(* IEC 61131-3 sources: ics-sorter-range/, 2 files *)

(* ---- Sorter.st ---- *)
(* Three-lane matrix sorter with nine trailer doors.
   Generated by gen_sorter.py. Do not hand edit; regenerate instead. *)

TYPE
  BELT_T : ARRAY[0..19] OF INT;
END_TYPE

PROGRAM sorter
VAR
  sorter_run    AT %QX110.0    : BOOL;   (* operator master run *)
  auto_mode     AT %QX110.1    : BOOL;   (* auto routing enabled *)
  lane1_run     AT %QX110.2    : BOOL;   (* induct 1 running *)
  lane2_run     AT %QX110.3    : BOOL;   (* induct 2 running *)
  lane3_run     AT %QX110.4    : BOOL;   (* induct 3 running *)
  ob1_run       AT %QX110.5    : BOOL;   (* outbound 1 running *)
  ob2_run       AT %QX110.6    : BOOL;   (* outbound 2 running *)
  ob3_run       AT %QX110.7    : BOOL;   (* outbound 3 running *)
  l1_div1       AT %QX111.0    : BOOL;   (* lane 1 divert to outbound 1 *)
  l1_div2       AT %QX111.1    : BOOL;   (* lane 1 divert to outbound 2 *)
  l1_div3       AT %QX111.2    : BOOL;   (* lane 1 divert to outbound 3 *)
  l2_div1       AT %QX111.3    : BOOL;   (* lane 2 divert to outbound 1 *)
  l2_div2       AT %QX111.4    : BOOL;   (* lane 2 divert to outbound 2 *)
  l2_div3       AT %QX111.5    : BOOL;   (* lane 2 divert to outbound 3 *)
  l3_div1       AT %QX111.6    : BOOL;   (* lane 3 divert to outbound 1 *)
  l3_div2       AT %QX111.7    : BOOL;   (* lane 3 divert to outbound 2 *)
  l3_div3       AT %QX112.0    : BOOL;   (* lane 3 divert to outbound 3 *)
  b1_door1      AT %QX112.1    : BOOL;   (* outbound 1 divert to door 1 *)
  b1_door2      AT %QX112.2    : BOOL;   (* outbound 1 divert to door 2 *)
  b1_door3      AT %QX112.3    : BOOL;   (* outbound 1 divert to door 3 *)
  b2_door1      AT %QX112.4    : BOOL;   (* outbound 2 divert to door 1 *)
  b2_door2      AT %QX112.5    : BOOL;   (* outbound 2 divert to door 2 *)
  b2_door3      AT %QX112.6    : BOOL;   (* outbound 2 divert to door 3 *)
  b3_door1      AT %QX112.7    : BOOL;   (* outbound 3 divert to door 1 *)
  b3_door2      AT %QX113.0    : BOOL;   (* outbound 3 divert to door 2 *)
  b3_door3      AT %QX113.1    : BOOL;   (* outbound 3 divert to door 3 *)
  jam_alarm     AT %QX113.2    : BOOL;   (* induct belt backing up at the tail *)
  coll_alarm    AT %QX113.3    : BOOL;   (* merge collision on an outbound belt *)
  noread_alarm  AT %QX113.4    : BOOL;   (* tunnel no-read *)
  nohome_alarm  AT %QX113.5    : BOOL;   (* package reached end of an outbound belt *)
  reset_cmd     AT %QX113.6    : BOOL;   (* re-run the init block, clearing all process state *)
  fault_reset   AT %QX113.7    : BOOL;   (* hold the drive fault-reset bit for several scans *)
  scanner_fault_ack AT %QX114.0 : BOOL; (* operator acknowledges scanner fault *)
  scanner_retry AT %QX114.1 : BOOL;     (* operator retries after acknowledgement *)
  xle_mode AT %QX114.2 : BOOL;           (* lane 1 external sort decisions *)
  xle_multi AT %QX114.3 : BOOL;          (* bounded two-package external mode *)
  plant_mode AT %QX114.6 : BOOL;          (* lane 1 position comes from drives plant *)
  photoeye_mode AT %QX114.7 : BOOL;       (* opt-in stateful field inputs; legacy events remain *)
  accumulation_mode AT %QX115.0 : BOOL;   (* opt-in finite plant zones; coil 920 *)

  speed_sp_1    AT %QW200      : INT;    (* induct 1 speed setpoint, rpm *)
  speed_sp_2    AT %QW201      : INT;    (* induct 2 speed setpoint, rpm *)
  speed_sp_3    AT %QW202      : INT;    (* induct 3 speed setpoint, rpm *)
  ob_speed_1    AT %QW203      : INT;    (* outbound 1 speed setpoint, rpm *)
  ob_speed_2    AT %QW204      : INT;    (* outbound 2 speed setpoint, rpm *)
  ob_speed_3    AT %QW205      : INT;    (* outbound 3 speed setpoint, rpm *)
  min_gap_sp    AT %QW206      : INT;    (* minimum induct gap, cells *)
  rate_sp_1     AT %QW207      : INT;    (* induct 1 interval, scans per package *)
  rate_sp_2     AT %QW208      : INT;    (* induct 2 interval, scans per package *)
  rate_sp_3     AT %QW209      : INT;    (* induct 3 interval, scans per package *)
  noread_sp     AT %QW210      : INT;    (* tunnel no-read rate, per mille *)
  scan_code_1   AT %QW211      : INT;    (* last barcode read by tunnel 1 *)
  scan_code_2   AT %QW212      : INT;    (* last barcode read by tunnel 2 *)
  scan_code_3   AT %QW213      : INT;    (* last barcode read by tunnel 3 *)
  noread_ct     AT %QW214      : INT;    (* cumulative tunnel no-reads *)
  coll_ct       AT %QW215      : INT;    (* cumulative merge collisions *)
  jam_ct        AT %QW216      : INT;    (* cumulative induct belt jams *)
  missort_ct    AT %QW217      : INT;    (* cumulative confirmed missorts at door scan *)
  recirc_ct     AT %QW218      : INT;    (* packages undiverted off an induct belt *)
  nohome_ct     AT %QW219      : INT;    (* packages undiverted off an outbound belt *)
  inducted_ct   AT %QW220      : INT;    (* cumulative packages inducted *)
  serial_next   AT %QW221      : INT;    (* next package serial number *)
  tr11_ct       AT %QW222      : INT;    (* packages loaded to trailer 1-1 *)
  tr12_ct       AT %QW223      : INT;    (* packages loaded to trailer 1-2 *)
  tr13_ct       AT %QW224      : INT;    (* packages loaded to trailer 1-3 *)
  tr21_ct       AT %QW225      : INT;    (* packages loaded to trailer 2-1 *)
  tr22_ct       AT %QW226      : INT;    (* packages loaded to trailer 2-2 *)
  tr23_ct       AT %QW227      : INT;    (* packages loaded to trailer 2-3 *)
  tr31_ct       AT %QW228      : INT;    (* packages loaded to trailer 3-1 *)
  tr32_ct       AT %QW229      : INT;    (* packages loaded to trailer 3-2 *)
  tr33_ct       AT %QW230      : INT;    (* packages loaded to trailer 3-3 *)
  tr11_bad      AT %QW231      : INT;    (* wrong-destination loads at trailer 1-1 *)
  tr12_bad      AT %QW232      : INT;    (* wrong-destination loads at trailer 1-2 *)
  tr13_bad      AT %QW233      : INT;    (* wrong-destination loads at trailer 1-3 *)
  tr21_bad      AT %QW234      : INT;    (* wrong-destination loads at trailer 2-1 *)
  tr22_bad      AT %QW235      : INT;    (* wrong-destination loads at trailer 2-2 *)
  tr23_bad      AT %QW236      : INT;    (* wrong-destination loads at trailer 2-3 *)
  tr31_bad      AT %QW237      : INT;    (* wrong-destination loads at trailer 3-1 *)
  tr32_bad      AT %QW238      : INT;    (* wrong-destination loads at trailer 3-2 *)
  tr33_bad      AT %QW239      : INT;    (* wrong-destination loads at trailer 3-3 *)
  div_act_1     AT %QW240      : INT;    (* outbound 1 induct-divert actuations *)
  div_act_2     AT %QW241      : INT;    (* outbound 2 induct-divert actuations *)
  div_act_3     AT %QW242      : INT;    (* outbound 3 induct-divert actuations *)
  scan_ct       AT %QW243      : INT;    (* PLC scans since init, logical clock *)
  shift_ct_1    AT %QW244      : INT;    (* induct 1 belt shifts since init *)
  shift_ct_2    AT %QW245      : INT;    (* induct 2 belt shifts since init *)
  shift_ct_3    AT %QW246      : INT;    (* induct 3 belt shifts since init *)
  master_seed   AT %QW247      : INT;    (* PRNG root, 1..999, 0 means use default *)
  run_id        AT %QW248      : INT;    (* scenario run identifier, echoed into telemetry *)
  prog_hash     AT %QW249      : INT;    (* identity of the generated program, set at init *)
  multiple_ct   AT %QW250      : INT;    (* tunnel reported more than one barcode *)
  oversize_ct   AT %QW251      : INT;    (* package exceeded the tunnel size limit *)
  duplicate_ct  AT %QW252      : INT;    (* tunnel returned a barcode already seen *)
  invalid_ct    AT %QW253      : INT;    (* tunnel decoded something that is not a label *)
  scan_late_ct  AT %QW254      : INT;    (* package left the tunnel before its result arrived *)
  scanner_state AT %QW255 : INT;        (* 0 ready, 1 prepare, 2 reset, 3 fault, 4 acknowledged *)
  scanner_fault_mask AT %QW256 : INT;   (* bits 0,1,2 identify missing tunnel ACKs *)
  scanner_ack_mask AT %QW257 : INT;     (* bits 0,1,2 for current phase ACKs *)
  scanner_wait AT %QW258 : INT;         (* elapsed PLC scans in current phase *)
  xle_cmd_id AT %QW500 : INT;            (* XLe writes 500..503 *)
  xle_cmd_bc AT %QW501 : INT;
  xle_cmd_dest AT %QW502 : INT;
  xle_cmd_nonce AT %QW503 : INT;
  xle_ack_id AT %QW504 : INT;            (* PLC writes 504..509 *)
  xle_state AT %QW505 : INT;             (* 0 idle, 1 accepted, 2 diverted, 3 loaded, 4 failed, 5 recirc *)
  xle_reason AT %QW506 : INT;            (* 1 no decision, 2 invalid/late, 3 collision, 4 no home, 5 wrong door *)
  xle_actual AT %QW507 : INT;            (* physical trailer, 1..9 *)
  xle_package AT %QW508 : INT;           (* scanner barcode identity *)
  xle_run_nonce AT %QW509 : INT;
  xle_scan_tick AT %QW510 : INT;          (* PLC scan accepting tunnel 1 result *)
  xle_accept_tick AT %QW511 : INT;        (* PLC scan accepting XLe command *)
  xle_divert_tick AT %QW512 : INT;        (* first arrival at lane 1 cell 14 *)
  multi_op AT %QW520 : INT;              (* 1 route, 2 release terminal slot *)
  multi_slot AT %QW521 : INT;            (* slot index 0..2 *)
  multi_token AT %QW522 : INT;
  multi_serial AT %QW523 : INT;
  multi_seq AT %QW524 : INT;
  multi_bc AT %QW525 : INT;
  multi_dest AT %QW526 : INT;
  multi_nonce AT %QW527 : INT;
  multi_cmd_id AT %QW528 : INT;          (* write last; changed ID commits payload *)
  multi_ack AT %QW529 : INT;             (* 1 accepted, 2 rejected, 3 released *)
  slot0_token AT %QW530 : INT;
  slot0_serial AT %QW531 : INT;
  slot0_seq AT %QW532 : INT;
  slot0_bc AT %QW533 : INT;
  slot0_state AT %QW534 : INT;
  slot0_dest AT %QW535 : INT;
  slot0_actual AT %QW536 : INT;
  slot0_reason AT %QW537 : INT;
  slot0_scan AT %QW538 : INT;
  slot0_accept AT %QW539 : INT;
  slot0_divert AT %QW540 : INT;
  slot0_command AT %QW541 : INT;
  slot1_token AT %QW542 : INT;
  slot1_serial AT %QW543 : INT;
  slot1_seq AT %QW544 : INT;
  slot1_bc AT %QW545 : INT;
  slot1_state AT %QW546 : INT;
  slot1_dest AT %QW547 : INT;
  slot1_actual AT %QW548 : INT;
  slot1_reason AT %QW549 : INT;
  slot1_scan AT %QW550 : INT;
  slot1_accept AT %QW551 : INT;
  slot1_divert AT %QW552 : INT;
  slot1_command AT %QW553 : INT;
  multi_ack_id AT %QW554 : INT;         (* PLC echoes processed command ID *)
  epoch_offer_lo AT %QW555 : INT;       (* XLe durable run ID, base 30000 *)
  epoch_offer_hi AT %QW556 : INT;
  epoch_offer_id AT %QW557 : INT;       (* write last to commit offer *)
  epoch_active_lo AT %QW558 : INT;      (* PLC accepted run ID *)
  epoch_active_hi AT %QW559 : INT;
  epoch_ack_id AT %QW560 : INT;
  epoch_fault AT %QW561 : INT;          (* 0 ready, 1 no identity, 2 XLe fault *)
  cmd_epoch_lo AT %QW562 : INT;
  cmd_epoch_hi AT %QW563 : INT;
  epoch_fault_request AT %QW564 : INT;  (* XLe 2 = fail closed *)
  hb_epoch_lo AT %QW565 : INT;          (* heartbeat payload before sequence *)
  hb_epoch_hi AT %QW566 : INT;
  hb_sequence AT %QW567 : INT;          (* XLe changes at least every 5 s *)
  hb_age AT %QW568 : INT;               (* PLC scans since valid heartbeat *)
  xle_liveness AT %QW569 : INT;         (* 0 healthy, 1 lost, 2 seen, 3 retry *)
  recovery_epoch_lo AT %QW570 : INT;
  recovery_epoch_hi AT %QW571 : INT;
  recovery_sequence AT %QW572 : INT;   (* XLe writes after journal verification *)
  hb_ack_sequence AT %QW573 : INT;
  plant_request AT %QW574 : INT;         (* PLC commits induction request last *)
  plant_request_token AT %QW575 : INT;
  plant_request_serial AT %QW576 : INT;
  plant_request_lane AT %QW577 : INT;   (* 1..3; written before request commit *)
  plant_event_lane AT %QW578 : INT;     (* plant payload, written before event commit *)
  plant_event_type AT %QW580 : INT;      (* 1 induct, 2 tunnel, 3 divert, 4 trailer, 5 recirc, 6 failed confirmation *)
  plant_event_token AT %QW581 : INT;
  plant_event_serial AT %QW582 : INT;
  plant_event_actual AT %QW583 : INT;    (* outbound 1..3 or trailer 1..9 *)
  plant_event_position AT %QW584 : INT;  (* tenths of a cell, telemetry *)
  plant_event_seq AT %QW585 : INT;       (* plant commits event last *)
  plant_event_ack AT %QW586 : INT;       (* PLC acknowledges even rejected events *)
  plant_epoch_lo AT %QW587 : INT;
  plant_epoch_hi AT %QW588 : INT;
  plant_nonce AT %QW589 : INT;
  plant_heartbeat AT %QW590 : INT;
  plant_fault AT %QW591 : INT;          (* 0 ready, 1 unavailable, 2 identity mismatch, 3 bad event *)
  plant_failed_count AT %QW592 : INT;   (* latched failed physical confirmations, cleared by reset *)
  plant_heartbeat_age AT %QW593 : INT;  (* PLC scans since the last plant heartbeat *)
  p0_raw_epoch_lo AT %QW600 : INT;
  p0_raw_epoch_hi AT %QW601 : INT;
  p0_raw_nonce AT %QW602 : INT;
  p0_raw_token AT %QW603 : INT;
  p0_raw_serial AT %QW604 : INT;
  p0_raw_belt AT %QW605 : INT;
  p0_raw_pos AT %QW606 : INT;
  p0_raw_event AT %QW607 : INT;
  p0_raw_actual AT %QW608 : INT;
  p0_raw_seq AT %QW609 : INT;
  p1_raw_epoch_lo AT %QW610 : INT;
  p1_raw_epoch_hi AT %QW611 : INT;
  p1_raw_nonce AT %QW612 : INT;
  p1_raw_token AT %QW613 : INT;
  p1_raw_serial AT %QW614 : INT;
  p1_raw_belt AT %QW615 : INT;
  p1_raw_pos AT %QW616 : INT;
  p1_raw_event AT %QW617 : INT;
  p1_raw_actual AT %QW618 : INT;
  p1_raw_seq AT %QW619 : INT;
  p0_view_epoch_lo AT %QW620 : INT;
  p0_view_epoch_hi AT %QW621 : INT;
  p0_view_nonce AT %QW622 : INT;
  p0_view_token AT %QW623 : INT;
  p0_view_serial AT %QW624 : INT;
  p0_view_belt AT %QW625 : INT;
  p0_view_pos AT %QW626 : INT;
  p0_view_event AT %QW627 : INT;
  p0_view_actual AT %QW628 : INT;
  p0_view_seq AT %QW629 : INT;
  p1_view_epoch_lo AT %QW630 : INT;
  p1_view_epoch_hi AT %QW631 : INT;
  p1_view_nonce AT %QW632 : INT;
  p1_view_token AT %QW633 : INT;
  p1_view_serial AT %QW634 : INT;
  p1_view_belt AT %QW635 : INT;
  p1_view_pos AT %QW636 : INT;
  p1_view_event AT %QW637 : INT;
  p1_view_actual AT %QW638 : INT;
  p1_view_seq AT %QW639 : INT;
  p0_view_status AT %QW640 : INT;       (* 0 empty, 1 live, 2 stale, 3 identity mismatch *)
  p1_view_status AT %QW641 : INT;
  p0_view_age AT %QW642 : INT;
  p1_view_age AT %QW643 : INT;
  slot0_lane AT %QW644 : INT;           (* stable lane identity beside slot row *)
  slot1_lane AT %QW645 : INT;
  plant_failed_lane AT %QW646 : INT;    (* lane of latest failed confirmation *)
  slot2_token AT %QW647 : INT;
  slot2_serial AT %QW648 : INT;
  slot2_seq AT %QW649 : INT;
  slot2_bc AT %QW650 : INT;
  slot2_state AT %QW651 : INT;
  slot2_dest AT %QW652 : INT;
  slot2_actual AT %QW653 : INT;
  slot2_reason AT %QW654 : INT;
  slot2_scan AT %QW655 : INT;
  slot2_accept AT %QW656 : INT;
  slot2_divert AT %QW657 : INT;
  slot2_command AT %QW658 : INT;
  slot2_lane AT %QW659 : INT;
  p2_raw_epoch_lo AT %QW660 : INT;
  p2_raw_epoch_hi AT %QW661 : INT;
  p2_raw_nonce AT %QW662 : INT;
  p2_raw_token AT %QW663 : INT;
  p2_raw_serial AT %QW664 : INT;
  p2_raw_belt AT %QW665 : INT;
  p2_raw_pos AT %QW666 : INT;
  p2_raw_event AT %QW667 : INT;
  p2_raw_actual AT %QW668 : INT;
  p2_raw_seq AT %QW669 : INT;
  p2_view_epoch_lo AT %QW670 : INT;
  p2_view_epoch_hi AT %QW671 : INT;
  p2_view_nonce AT %QW672 : INT;
  p2_view_token AT %QW673 : INT;
  p2_view_serial AT %QW674 : INT;
  p2_view_belt AT %QW675 : INT;
  p2_view_pos AT %QW676 : INT;
  p2_view_event AT %QW677 : INT;
  p2_view_actual AT %QW678 : INT;
  p2_view_seq AT %QW679 : INT;
  p2_view_status AT %QW680 : INT;
  p2_view_age AT %QW681 : INT;
  pe0_raw_epoch_lo AT %QW690 : INT;
  pe0_raw_epoch_hi AT %QW691 : INT;
  pe0_raw_nonce AT %QW692 : INT;
  pe0_raw_token AT %QW693 : INT;
  pe0_raw_serial AT %QW694 : INT;
  pe0_raw_lane AT %QW695 : INT;
  pe0_raw_mask AT %QW696 : INT;          (* bits 0..4: induct,tunnel,divert,outbound,trailer *)
  pe0_raw_seq AT %QW697 : INT;           (* plant commits the complete row last *)
  pe1_raw_epoch_lo AT %QW698 : INT;
  pe1_raw_epoch_hi AT %QW699 : INT;
  pe1_raw_nonce AT %QW700 : INT;
  pe1_raw_token AT %QW701 : INT;
  pe1_raw_serial AT %QW702 : INT;
  pe1_raw_lane AT %QW703 : INT;
  pe1_raw_mask AT %QW704 : INT;
  pe1_raw_seq AT %QW705 : INT;
  pe2_raw_epoch_lo AT %QW706 : INT;
  pe2_raw_epoch_hi AT %QW707 : INT;
  pe2_raw_nonce AT %QW708 : INT;
  pe2_raw_token AT %QW709 : INT;
  pe2_raw_serial AT %QW710 : INT;
  pe2_raw_lane AT %QW711 : INT;
  pe2_raw_mask AT %QW712 : INT;
  pe2_raw_seq AT %QW713 : INT;
  pe0_view_epoch_lo AT %QW720 : INT;
  pe0_view_epoch_hi AT %QW721 : INT;
  pe0_view_nonce AT %QW722 : INT;
  pe0_view_token AT %QW723 : INT;
  pe0_view_serial AT %QW724 : INT;
  pe0_view_raw AT %QW725 : INT;
  pe0_view_conditioned AT %QW726 : INT;
  pe0_view_quality AT %QW727 : INT;
  pe1_view_epoch_lo AT %QW728 : INT;
  pe1_view_epoch_hi AT %QW729 : INT;
  pe1_view_nonce AT %QW730 : INT;
  pe1_view_token AT %QW731 : INT;
  pe1_view_serial AT %QW732 : INT;
  pe1_view_raw AT %QW733 : INT;
  pe1_view_conditioned AT %QW734 : INT;
  pe1_view_quality AT %QW735 : INT;
  pe2_view_epoch_lo AT %QW736 : INT;
  pe2_view_epoch_hi AT %QW737 : INT;
  pe2_view_nonce AT %QW738 : INT;
  pe2_view_token AT %QW739 : INT;
  pe2_view_serial AT %QW740 : INT;
  pe2_view_raw AT %QW741 : INT;
  pe2_view_conditioned AT %QW742 : INT;
  pe2_view_quality AT %QW743 : INT;
  pe_debounce_sp AT %QW744 : INT;         (* 1..5 PLC scans *)
  pe_min_block_sp AT %QW745 : INT;       (* 1..30 PLC scans *)
  pe_max_block_sp AT %QW746 : INT;       (* 2..300 PLC scans *)
  pe_travel_sp AT %QW747 : INT;          (* 5..1000 PLC scans *)
  pe_fault_mask AT %QW748 : INT;         (* bit per occupied slot, latched to reset *)
  pe_fault_sensor AT %QW749 : INT;       (* 1..5 latest failed photoeye *)
  pe_fault_lane AT %QW750 : INT;
  z0_raw_zone AT %QW751 : INT;
  z0_raw_motion AT %QW752 : INT;
  z0_raw_hold AT %QW753 : INT;
  z0_raw_dwell AT %QW754 : INT;
  z0_raw_seq AT %QW755 : INT;
  z1_raw_zone AT %QW756 : INT;
  z1_raw_motion AT %QW757 : INT;
  z1_raw_hold AT %QW758 : INT;
  z1_raw_dwell AT %QW759 : INT;
  z1_raw_seq AT %QW760 : INT;
  z2_raw_zone AT %QW761 : INT;
  z2_raw_motion AT %QW762 : INT;
  z2_raw_hold AT %QW763 : INT;
  z2_raw_dwell AT %QW764 : INT;
  z2_raw_seq AT %QW765 : INT;
  z0_view_zone AT %QW766 : INT;
  z0_view_motion AT %QW767 : INT;
  z0_view_hold AT %QW768 : INT;
  z0_view_dwell AT %QW769 : INT;
  z0_view_seq AT %QW770 : INT;
  z1_view_zone AT %QW771 : INT;
  z1_view_motion AT %QW772 : INT;
  z1_view_hold AT %QW773 : INT;
  z1_view_dwell AT %QW774 : INT;
  z1_view_seq AT %QW775 : INT;
  z2_view_zone AT %QW776 : INT;
  z2_view_motion AT %QW777 : INT;
  z2_view_hold AT %QW778 : INT;
  z2_view_dwell AT %QW779 : INT;
  z2_view_seq AT %QW780 : INT;
  z0_quality AT %QW781 : INT;          (* 0 empty, 1 valid, 2 stale, 3 rejected *)
  z1_quality AT %QW782 : INT;
  z2_quality AT %QW783 : INT;
  z_raw_ready AT %QW784 : INT;         (* plant capacity mask, bits 0..2 *)
  z_raw_commit AT %QW785 : INT;        (* plant heartbeat, written after all rows *)
  z_view_ready AT %QW786 : INT;        (* PLC-accepted capacity mask *)
  z_view_age AT %QW787 : INT;
  z_fault AT %QW788 : INT;             (* 0 ready, 1 identity/sequence, 2 bounds/order, 3 overlap *)
  chute_mode AT %QX115.1 : BOOL;        (* coil 921, selected chute opt-in *)
  chute_raw_version AT %QW790 : INT;
  chute_raw_trailer AT %QW791 : INT;
  chute_raw_occupied AT %QW792 : INT;
  chute_raw_reserved AT %QW793 : INT;
  chute_raw_full AT %QW794 : INT;
  chute_raw_epoch_lo AT %QW795 : INT;
  chute_raw_epoch_hi AT %QW796 : INT;
  chute_raw_nonce AT %QW797 : INT;
  chute_raw_seq AT %QW798 : INT;
  chute_raw_token AT %QW799 : INT;
  chute_raw_serial AT %QW800 : INT;
  chute_raw_event_seq AT %QW801 : INT;
  chute_raw_commit AT %QW802 : INT;
  chute_raw_ack AT %QW803 : INT;
  chute_view_trailer AT %QW804 : INT;
  chute_view_occupied AT %QW805 : INT;
  chute_state AT %QW806 : INT;
  chute_quality AT %QW807 : INT;
  chute_age AT %QW808 : INT;
  chute_permissive AT %QW809 : INT;
  chute_empty_trailer AT %QW810 : INT;
  chute_empty_epoch_lo AT %QW811 : INT;
  chute_empty_epoch_hi AT %QW812 : INT;
  chute_empty_nonce AT %QW813 : INT;
  chute_empty_seq AT %QW814 : INT;
  chute_empty_result AT %QW815 : INT;
  chute_empty_ack AT %QW816 : INT;
  chute_action_trailer AT %QW817 : INT;
  chute_action_epoch_lo AT %QW818 : INT;
  chute_action_epoch_hi AT %QW819 : INT;
  chute_action_nonce AT %QW820 : INT;
  chute_action_op AT %QW821 : INT;
  chute_action_seq AT %QW822 : INT;
  chute_action_ack AT %QW823 : INT;
  chute_action_result AT %QW824 : INT;
  chute_config_trailer AT %QW825 : INT;
  chute_config_capacity AT %QW826 : INT;
  chute_accepted_token AT %QW827 : INT;
  chute_accepted_serial AT %QW828 : INT;
  chute_accepted_event_seq AT %QW829 : INT;
  chute_raw_accepted_token AT %QW830 : INT;
  chute_raw_accepted_serial AT %QW831 : INT;
  chute_raw_accepted_seq AT %QW832 : INT;
  xle_fault_ack AT %QX114.4 : BOOL;    (* coil 916, operator action *)
  xle_retry AT %QX114.5 : BOOL;        (* coil 917, operator action *)

  ib1_c0          AT %QW260      : INT;
  ib1_c1          AT %QW261      : INT;
  ib1_c2          AT %QW262      : INT;
  ib1_c3          AT %QW263      : INT;
  ib1_c4          AT %QW264      : INT;
  ib1_c5          AT %QW265      : INT;
  ib1_c6          AT %QW266      : INT;
  ib1_c7          AT %QW267      : INT;
  ib1_c8          AT %QW268      : INT;
  ib1_c9          AT %QW269      : INT;
  ib1_c10         AT %QW270      : INT;
  ib1_c11         AT %QW271      : INT;
  ib1_c12         AT %QW272      : INT;
  ib1_c13         AT %QW273      : INT;
  ib1_c14         AT %QW274      : INT;
  ib1_c15         AT %QW275      : INT;
  ib1_c16         AT %QW276      : INT;
  ib1_c17         AT %QW277      : INT;
  ib1_c18         AT %QW278      : INT;
  ib1_c19         AT %QW279      : INT;
  ib2_c0          AT %QW280      : INT;
  ib2_c1          AT %QW281      : INT;
  ib2_c2          AT %QW282      : INT;
  ib2_c3          AT %QW283      : INT;
  ib2_c4          AT %QW284      : INT;
  ib2_c5          AT %QW285      : INT;
  ib2_c6          AT %QW286      : INT;
  ib2_c7          AT %QW287      : INT;
  ib2_c8          AT %QW288      : INT;
  ib2_c9          AT %QW289      : INT;
  ib2_c10         AT %QW290      : INT;
  ib2_c11         AT %QW291      : INT;
  ib2_c12         AT %QW292      : INT;
  ib2_c13         AT %QW293      : INT;
  ib2_c14         AT %QW294      : INT;
  ib2_c15         AT %QW295      : INT;
  ib2_c16         AT %QW296      : INT;
  ib2_c17         AT %QW297      : INT;
  ib2_c18         AT %QW298      : INT;
  ib2_c19         AT %QW299      : INT;
  ib3_c0          AT %QW300      : INT;
  ib3_c1          AT %QW301      : INT;
  ib3_c2          AT %QW302      : INT;
  ib3_c3          AT %QW303      : INT;
  ib3_c4          AT %QW304      : INT;
  ib3_c5          AT %QW305      : INT;
  ib3_c6          AT %QW306      : INT;
  ib3_c7          AT %QW307      : INT;
  ib3_c8          AT %QW308      : INT;
  ib3_c9          AT %QW309      : INT;
  ib3_c10         AT %QW310      : INT;
  ib3_c11         AT %QW311      : INT;
  ib3_c12         AT %QW312      : INT;
  ib3_c13         AT %QW313      : INT;
  ib3_c14         AT %QW314      : INT;
  ib3_c15         AT %QW315      : INT;
  ib3_c16         AT %QW316      : INT;
  ib3_c17         AT %QW317      : INT;
  ib3_c18         AT %QW318      : INT;
  ib3_c19         AT %QW319      : INT;

  rt1_c0          AT %QW320      : INT;
  rt1_c1          AT %QW321      : INT;
  rt1_c2          AT %QW322      : INT;
  rt1_c3          AT %QW323      : INT;
  rt1_c4          AT %QW324      : INT;
  rt1_c5          AT %QW325      : INT;
  rt1_c6          AT %QW326      : INT;
  rt1_c7          AT %QW327      : INT;
  rt1_c8          AT %QW328      : INT;
  rt1_c9          AT %QW329      : INT;
  rt1_c10         AT %QW330      : INT;
  rt1_c11         AT %QW331      : INT;
  rt1_c12         AT %QW332      : INT;
  rt1_c13         AT %QW333      : INT;
  rt1_c14         AT %QW334      : INT;
  rt1_c15         AT %QW335      : INT;
  rt1_c16         AT %QW336      : INT;
  rt1_c17         AT %QW337      : INT;
  rt1_c18         AT %QW338      : INT;
  rt1_c19         AT %QW339      : INT;
  rt2_c0          AT %QW340      : INT;
  rt2_c1          AT %QW341      : INT;
  rt2_c2          AT %QW342      : INT;
  rt2_c3          AT %QW343      : INT;
  rt2_c4          AT %QW344      : INT;
  rt2_c5          AT %QW345      : INT;
  rt2_c6          AT %QW346      : INT;
  rt2_c7          AT %QW347      : INT;
  rt2_c8          AT %QW348      : INT;
  rt2_c9          AT %QW349      : INT;
  rt2_c10         AT %QW350      : INT;
  rt2_c11         AT %QW351      : INT;
  rt2_c12         AT %QW352      : INT;
  rt2_c13         AT %QW353      : INT;
  rt2_c14         AT %QW354      : INT;
  rt2_c15         AT %QW355      : INT;
  rt2_c16         AT %QW356      : INT;
  rt2_c17         AT %QW357      : INT;
  rt2_c18         AT %QW358      : INT;
  rt2_c19         AT %QW359      : INT;
  rt3_c0          AT %QW360      : INT;
  rt3_c1          AT %QW361      : INT;
  rt3_c2          AT %QW362      : INT;
  rt3_c3          AT %QW363      : INT;
  rt3_c4          AT %QW364      : INT;
  rt3_c5          AT %QW365      : INT;
  rt3_c6          AT %QW366      : INT;
  rt3_c7          AT %QW367      : INT;
  rt3_c8          AT %QW368      : INT;
  rt3_c9          AT %QW369      : INT;
  rt3_c10         AT %QW370      : INT;
  rt3_c11         AT %QW371      : INT;
  rt3_c12         AT %QW372      : INT;
  rt3_c13         AT %QW373      : INT;
  rt3_c14         AT %QW374      : INT;
  rt3_c15         AT %QW375      : INT;
  rt3_c16         AT %QW376      : INT;
  rt3_c17         AT %QW377      : INT;
  rt3_c18         AT %QW378      : INT;
  rt3_c19         AT %QW379      : INT;

  ob1_c0          AT %QW380      : INT;
  ob1_c1          AT %QW381      : INT;
  ob1_c2          AT %QW382      : INT;
  ob1_c3          AT %QW383      : INT;
  ob1_c4          AT %QW384      : INT;
  ob1_c5          AT %QW385      : INT;
  ob1_c6          AT %QW386      : INT;
  ob1_c7          AT %QW387      : INT;
  ob1_c8          AT %QW388      : INT;
  ob1_c9          AT %QW389      : INT;
  ob1_c10         AT %QW390      : INT;
  ob1_c11         AT %QW391      : INT;
  ob1_c12         AT %QW392      : INT;
  ob1_c13         AT %QW393      : INT;
  ob1_c14         AT %QW394      : INT;
  ob1_c15         AT %QW395      : INT;
  ob1_c16         AT %QW396      : INT;
  ob1_c17         AT %QW397      : INT;
  ob1_c18         AT %QW398      : INT;
  ob1_c19         AT %QW399      : INT;
  ob2_c0          AT %QW400      : INT;
  ob2_c1          AT %QW401      : INT;
  ob2_c2          AT %QW402      : INT;
  ob2_c3          AT %QW403      : INT;
  ob2_c4          AT %QW404      : INT;
  ob2_c5          AT %QW405      : INT;
  ob2_c6          AT %QW406      : INT;
  ob2_c7          AT %QW407      : INT;
  ob2_c8          AT %QW408      : INT;
  ob2_c9          AT %QW409      : INT;
  ob2_c10         AT %QW410      : INT;
  ob2_c11         AT %QW411      : INT;
  ob2_c12         AT %QW412      : INT;
  ob2_c13         AT %QW413      : INT;
  ob2_c14         AT %QW414      : INT;
  ob2_c15         AT %QW415      : INT;
  ob2_c16         AT %QW416      : INT;
  ob2_c17         AT %QW417      : INT;
  ob2_c18         AT %QW418      : INT;
  ob2_c19         AT %QW419      : INT;
  ob3_c0          AT %QW420      : INT;
  ob3_c1          AT %QW421      : INT;
  ob3_c2          AT %QW422      : INT;
  ob3_c3          AT %QW423      : INT;
  ob3_c4          AT %QW424      : INT;
  ob3_c5          AT %QW425      : INT;
  ob3_c6          AT %QW426      : INT;
  ob3_c7          AT %QW427      : INT;
  ob3_c8          AT %QW428      : INT;
  ob3_c9          AT %QW429      : INT;
  ob3_c10         AT %QW430      : INT;
  ob3_c11         AT %QW431      : INT;
  ob3_c12         AT %QW432      : INT;
  ob3_c13         AT %QW433      : INT;
  ob3_c14         AT %QW434      : INT;
  ob3_c15         AT %QW435      : INT;
  ob3_c16         AT %QW436      : INT;
  ob3_c17         AT %QW437      : INT;
  ob3_c18         AT %QW438      : INT;
  ob3_c19         AT %QW439      : INT;

  ort1_c0         AT %QW440      : INT;
  ort1_c1         AT %QW441      : INT;
  ort1_c2         AT %QW442      : INT;
  ort1_c3         AT %QW443      : INT;
  ort1_c4         AT %QW444      : INT;
  ort1_c5         AT %QW445      : INT;
  ort1_c6         AT %QW446      : INT;
  ort1_c7         AT %QW447      : INT;
  ort1_c8         AT %QW448      : INT;
  ort1_c9         AT %QW449      : INT;
  ort1_c10        AT %QW450      : INT;
  ort1_c11        AT %QW451      : INT;
  ort1_c12        AT %QW452      : INT;
  ort1_c13        AT %QW453      : INT;
  ort1_c14        AT %QW454      : INT;
  ort1_c15        AT %QW455      : INT;
  ort1_c16        AT %QW456      : INT;
  ort1_c17        AT %QW457      : INT;
  ort1_c18        AT %QW458      : INT;
  ort1_c19        AT %QW459      : INT;
  ort2_c0         AT %QW460      : INT;
  ort2_c1         AT %QW461      : INT;
  ort2_c2         AT %QW462      : INT;
  ort2_c3         AT %QW463      : INT;
  ort2_c4         AT %QW464      : INT;
  ort2_c5         AT %QW465      : INT;
  ort2_c6         AT %QW466      : INT;
  ort2_c7         AT %QW467      : INT;
  ort2_c8         AT %QW468      : INT;
  ort2_c9         AT %QW469      : INT;
  ort2_c10        AT %QW470      : INT;
  ort2_c11        AT %QW471      : INT;
  ort2_c12        AT %QW472      : INT;
  ort2_c13        AT %QW473      : INT;
  ort2_c14        AT %QW474      : INT;
  ort2_c15        AT %QW475      : INT;
  ort2_c16        AT %QW476      : INT;
  ort2_c17        AT %QW477      : INT;
  ort2_c18        AT %QW478      : INT;
  ort2_c19        AT %QW479      : INT;
  ort3_c0         AT %QW480      : INT;
  ort3_c1         AT %QW481      : INT;
  ort3_c2         AT %QW482      : INT;
  ort3_c3         AT %QW483      : INT;
  ort3_c4         AT %QW484      : INT;
  ort3_c5         AT %QW485      : INT;
  ort3_c6         AT %QW486      : INT;
  ort3_c7         AT %QW487      : INT;
  ort3_c8         AT %QW488      : INT;
  ort3_c9         AT %QW489      : INT;
  ort3_c10        AT %QW490      : INT;
  ort3_c11        AT %QW491      : INT;
  ort3_c12        AT %QW492      : INT;
  ort3_c13        AT %QW493      : INT;
  ort3_c14        AT %QW494      : INT;
  ort3_c15        AT %QW495      : INT;
  ort3_c16        AT %QW496      : INT;
  ort3_c17        AT %QW497      : INT;
  ort3_c18        AT %QW498      : INT;
  ort3_c19        AT %QW499      : INT;

  induct1_cmd  AT %QW100      : INT;
  induct1_ref  AT %QW101      : INT;
  induct1_load AT %QW102      : INT;
  induct1_fb   AT %IW105      : INT;
  induct2_cmd  AT %QW103      : INT;
  induct2_ref  AT %QW104      : INT;
  induct2_load AT %QW105      : INT;
  induct2_fb   AT %IW114      : INT;
  induct3_cmd  AT %QW106      : INT;
  induct3_ref  AT %QW107      : INT;
  induct3_load AT %QW108      : INT;
  induct3_fb   AT %IW123      : INT;
  outbnd1_cmd  AT %QW109      : INT;
  outbnd1_ref  AT %QW110      : INT;
  outbnd1_load AT %QW111      : INT;
  outbnd1_fb   AT %IW132      : INT;
  outbnd2_cmd  AT %QW112      : INT;
  outbnd2_ref  AT %QW113      : INT;
  outbnd2_load AT %QW114      : INT;
  outbnd2_fb   AT %IW141      : INT;
  outbnd3_cmd  AT %QW115      : INT;
  outbnd3_ref  AT %QW116      : INT;
  outbnd3_load AT %QW117      : INT;
  outbnd3_fb   AT %IW150      : INT;
  scan1_trig   AT %QW118      : INT;
  scan1_serial AT %QW119      : INT;
  scan1_seed   AT %QW120      : INT;
  scan1_nrrate AT %QW121      : INT;
  scan1_result AT %IW158      : INT;
  scan1_bc     AT %IW159      : INT;
  scan1_status AT %IW160      : INT;
  scan1_len    AT %IW161      : INT;
  scan1_nonce  AT %IW164      : INT;
  scan2_trig   AT %QW122      : INT;
  scan2_serial AT %QW123      : INT;
  scan2_seed   AT %QW124      : INT;
  scan2_nrrate AT %QW125      : INT;
  scan2_result AT %IW169      : INT;
  scan2_bc     AT %IW170      : INT;
  scan2_status AT %IW171      : INT;
  scan2_len    AT %IW172      : INT;
  scan2_nonce  AT %IW175      : INT;
  scan3_trig   AT %QW126      : INT;
  scan3_serial AT %QW127      : INT;
  scan3_seed   AT %QW128      : INT;
  scan3_nrrate AT %QW129      : INT;
  scan3_result AT %IW180      : INT;
  scan3_bc     AT %IW181      : INT;
  scan3_status AT %IW182      : INT;
  scan3_len    AT %IW183      : INT;
  scan3_nonce  AT %IW186      : INT;
END_VAR

VAR
  ib1 : BELT_T;
  ib2 : BELT_T;
  ib3 : BELT_T;
  rt1 : BELT_T;
  rt2 : BELT_T;
  rt3 : BELT_T;
  ob1 : BELT_T;
  ob2 : BELT_T;
  ob3 : BELT_T;
  ort1 : BELT_T;
  ort2 : BELT_T;
  ort3 : BELT_T;
  tok1, otok1, otok2, otok3 : BELT_T;
  st_token, st_serial, st_seq, st_bc : ARRAY[0..2] OF INT;
  st_lane : ARRAY[0..2] OF INT;
  st_state, st_dest, st_actual, st_reason : ARRAY[0..2] OF INT;
  st_scan, st_accept, st_divert, st_command : ARRAY[0..2] OF INT;
  acc_i1, acc_i2, acc_i3 : REAL := 0.0;
  acc_o1, acc_o2, acc_o3 : REAL := 0.0;
  tmr1, tmr2, tmr3 : INT := 0;
  last_tun_1, last_tun_2, last_tun_3 : INT := 0;
  i, dest, obelt, door, bc, occ : INT;
  jam_lat_1, jam_lat_2, jam_lat_3 : BOOL := FALSE;
  sts       : INT := 0;
  frst_tmr  : INT := 0;
  tun_pkg_1, tun_pkg_2, tun_pkg_3 : INT := 0;
  tun_seq_1, tun_seq_2, tun_seq_3 : INT := 0;
  tun_wait_1, tun_wait_2, tun_wait_3 : BOOL := FALSE;
  init_done : BOOL := FALSE;
  reset_nonce : INT := 0;
  xle_cmd_seen, xle_route_dest : INT := 0;
  xle_inducted : BOOL := FALSE;
  token_next, multi_seen, slot_index, j : INT := 0;
  epoch_offer_seen : INT := 0;
  hb_seen, recovery_seen : INT := 0;
  hb_ready : BOOL := FALSE;
  plant_seen, plant_hb_seen, plant_hb_age, plant_scan_token, plant_scan_token_2,
  plant_scan_token_3 : INT := 0;
  plant_request_pending : BOOL := FALSE;
  plant_lane_match : BOOL := FALSE;
  plant_next_lane : INT := 1;
  plant_pick_lane, plant_candidate : INT := 0;
  plant_view_seen0, plant_view_seen1, plant_view_seen2 : INT := 0;
  pe_bound_token, pe_seen, pe_age, pe_raw, pe_filtered,
  pe_quality, pe_expected, pe_travel : ARRAY[0..2] OF INT;
  pe_candidate, pe_duration : ARRAY[0..14] OF INT;
  pe_stable : ARRAY[0..14] OF BOOL;
  pe_epoch_lo, pe_epoch_hi, pe_nonce, pe_token,
  pe_serial, pe_lane, pe_mask, pe_seq : ARRAY[0..2] OF INT;
  pe_bit, pe_index, pe_sensor, pe_debounce, pe_min_block,
  pe_max_block, pe_max_travel : INT := 0;
  pe_is_raw, pe_event_ready : BOOL := FALSE;
  z_raw_zone, z_raw_motion, z_raw_hold, z_raw_dwell, z_raw_seq : ARRAY[0..2] OF INT;
  z_view_zone, z_view_motion, z_view_hold, z_view_dwell,
  z_view_seq, z_quality, z_bound_token : ARRAY[0..2] OF INT;
  z_belt, z_pos : ARRAY[0..2] OF INT;
  z_seen_commit, z_lane, z_difference : INT := 0;
  z_valid : BOOL := FALSE;
  chute_seen, chute_expect, chute_action_seen, chute_action_expect : INT := 0;
  chute_empty_next : INT := 0;
  chute_resume_grace : INT := 0; (* bounded committed hold sample at Resume *)
  chute_identity_ok, chute_valid : BOOL := FALSE;
  chute_accounted_token, chute_accounted_serial, chute_accounted_seq : INT := 0;
END_VAR

(* reset: clears init_done so the block below re-runs this scan *)
IF reset_cmd AND scanner_state = 0 THEN
  init_done := FALSE;
END_IF;
reset_cmd := FALSE;

IF NOT init_done THEN
  speed_sp_1 := 200; speed_sp_2 := 200; speed_sp_3 := 200;
  ob_speed_1 := 233; ob_speed_2 := 233; ob_speed_3 := 233;
  min_gap_sp := 2;
  rate_sp_1  := 14; rate_sp_2 := 14; rate_sp_3 := 14;
  noread_sp  := 30;
  serial_next := 1;
  prog_hash := 24115;

  (* master_seed is the root of the run. The controller no longer draws
     destinations or no-reads itself: both moved to the camera tunnels,
     which are seeded from this value. It is kept and forwarded rather
     than used here. *)
  IF master_seed <= 0 OR master_seed > 999 THEN
    master_seed := 137;
  END_IF;

  (* clear process state. Without this a reset would leave packages on
     the belts and counters mid-run, and replay would not be replay. *)
  scan_ct := 0;
  shift_ct_1 := 0;
  shift_ct_2 := 0;
  shift_ct_3 := 0;
  noread_ct := 0; coll_ct := 0; jam_ct := 0; missort_ct := 0;
  recirc_ct := 0; nohome_ct := 0; inducted_ct := 0;
  div_act_1 := 0;
  div_act_2 := 0;
  div_act_3 := 0;
  scan_code_1 := 0;
  xle_mode := FALSE;
  xle_multi := FALSE;
  plant_mode := FALSE;
  photoeye_mode := FALSE;
  accumulation_mode := FALSE;
  z_raw_ready := 0; z_view_ready := 0; z_view_age := 0;
  z_seen_commit := z_raw_commit; z_fault := 0;
  chute_mode := FALSE; chute_config_trailer := 2; chute_config_capacity := 3;
  chute_seen := 0; chute_raw_ack := 0; chute_view_trailer := 0;
  chute_view_occupied := 0; chute_state := 0; chute_quality := 0;
  chute_age := 0; chute_permissive := 1;
  chute_action_seen := chute_action_seq; chute_action_ack := 0;
  chute_action_result := 0; chute_empty_next := 0;
  chute_resume_grace := 0;
  chute_empty_seq := 0; chute_empty_result := 0; chute_empty_ack := 0;
  chute_accepted_token := 0; chute_accepted_serial := 0;
  chute_accepted_event_seq := 0;
  chute_accounted_token := 0; chute_accounted_serial := 0;
  chute_accounted_seq := 0;
  pe_debounce_sp := 2; pe_min_block_sp := 2;
  pe_max_block_sp := 120; pe_travel_sp := 400;
  pe_fault_mask := 0; pe_fault_sensor := 0; pe_fault_lane := 0;
  plant_request := 0; plant_request_token := 0; plant_request_serial := 0;
  plant_request_lane := 0;
  plant_seen := plant_event_seq; plant_event_ack := 0;
  plant_hb_seen := plant_heartbeat; plant_hb_age := 0;
  plant_scan_token := 0; plant_scan_token_2 := 0; plant_scan_token_3 := 0;
  plant_request_pending := FALSE; plant_fault := 1;
  plant_next_lane := 1;
  plant_failed_count := 0;
  plant_failed_lane := 0;
  plant_heartbeat_age := 0;
  plant_view_seen0 := p0_raw_seq; plant_view_seen1 := p1_raw_seq;
  plant_view_seen2 := p2_raw_seq;
  p0_view_status := 0; p1_view_status := 0; p2_view_status := 0;
  p0_view_age := 0; p1_view_age := 0; p2_view_age := 0;
  p0_view_token := 0; p1_view_token := 0; p2_view_token := 0;
  p0_view_belt := 0; p1_view_belt := 0; p2_view_belt := 0;
  slot0_lane := 0; slot1_lane := 0; slot2_lane := 0;
  multi_seen := multi_cmd_id; multi_ack := 0; multi_ack_id := 0; token_next := 0;
  epoch_offer_seen := epoch_offer_id; epoch_ack_id := 0;
  epoch_active_lo := 0; epoch_active_hi := 0; epoch_fault := 1;
  epoch_fault_request := 0;
  hb_seen := hb_sequence; hb_ack_sequence := 0;
  hb_age := 0; hb_ready := FALSE; xle_liveness := 0;
  recovery_seen := recovery_sequence;
  xle_fault_ack := FALSE; xle_retry := FALSE;
  FOR j := 0 TO 2 DO
    st_token[j] := 0; st_serial[j] := 0; st_seq[j] := 0; st_bc[j] := 0;
    st_lane[j] := 0;
    st_state[j] := 0; st_dest[j] := 0; st_actual[j] := 0;
    st_reason[j] := 0; st_scan[j] := 0; st_accept[j] := 0;
    st_divert[j] := 0; st_command[j] := 0;
    pe_bound_token[j] := 0; pe_seen[j] := 0; pe_age[j] := 0;
    pe_raw[j] := 0; pe_filtered[j] := 0; pe_quality[j] := 0;
    pe_expected[j] := 1; pe_travel[j] := 0;
    z_bound_token[j] := 0; z_view_zone[j] := 0;
    z_view_motion[j] := 0; z_view_hold[j] := 0;
    z_view_dwell[j] := 0; z_view_seq[j] := 0;
    z_quality[j] := 0;
  END_FOR;
  FOR j := 0 TO 14 DO
    pe_candidate[j] := 0; pe_duration[j] := 0; pe_stable[j] := FALSE;
  END_FOR;
  pe0_view_token := 0; pe0_view_raw := 0; pe0_view_conditioned := 0; pe0_view_quality := 0;
  pe1_view_token := 0; pe1_view_raw := 0; pe1_view_conditioned := 0; pe1_view_quality := 0;
  pe2_view_token := 0; pe2_view_raw := 0; pe2_view_conditioned := 0; pe2_view_quality := 0;
  xle_cmd_seen := xle_cmd_id;
  xle_route_dest := 0;
  xle_inducted := FALSE;
  xle_ack_id := 0; xle_state := 0; xle_reason := 0;
  xle_actual := 0; xle_package := 0;
  xle_scan_tick := 0; xle_accept_tick := 0; xle_divert_tick := 0;
  acc_i1 := 0.0; tmr1 := 0; jam_lat_1 := FALSE;
  acc_o1 := 0.0;
  scan_code_2 := 0;
  acc_i2 := 0.0; tmr2 := 0; jam_lat_2 := FALSE;
  acc_o2 := 0.0;
  scan_code_3 := 0;
  acc_i3 := 0.0; tmr3 := 0; jam_lat_3 := FALSE;
  acc_o3 := 0.0;
  tr11_ct := 0; tr11_bad := 0;
  tr12_ct := 0; tr12_bad := 0;
  tr13_ct := 0; tr13_bad := 0;
  tr21_ct := 0; tr21_bad := 0;
  tr22_ct := 0; tr22_bad := 0;
  tr23_ct := 0; tr23_bad := 0;
  tr31_ct := 0; tr31_bad := 0;
  tr32_ct := 0; tr32_bad := 0;
  tr33_ct := 0; tr33_bad := 0;
  FOR i := 0 TO 19 DO
    ib1[i] := 0; rt1[i] := 0; tok1[i] := 0;
    ob1[i] := 0; ort1[i] := 0; otok1[i] := 0;
    ib2[i] := 0; rt2[i] := 0;
    ob2[i] := 0; ort2[i] := 0; otok2[i] := 0;
    ib3[i] := 0; rt3[i] := 0;
    ob3[i] := 0; ort3[i] := 0; otok3[i] := 0;
  END_FOR;
  induct1_load := 0;
  induct2_load := 0;
  induct3_load := 0;
  outbnd1_load := 0;
  outbnd2_load := 0;
  outbnd3_load := 0;
  frst_tmr := 0;
  multiple_ct := 0; oversize_ct := 0; duplicate_ct := 0;
  invalid_ct := 0; scan_late_ct := 0;
  tun_pkg_1 := 0; tun_seq_1 := 0; tun_wait_1 := FALSE;
  tun_pkg_2 := 0; tun_seq_2 := 0; tun_wait_2 := FALSE;
  tun_pkg_3 := 0; tun_seq_3 := 0; tun_wait_3 := FALSE;
  reset_nonce := reset_nonce + 1;
  IF reset_nonce > 30000 THEN reset_nonce := 1; END_IF;
  xle_run_nonce := reset_nonce;
  scanner_state := 1; scanner_wait := 0;
  scanner_fault_mask := 0; scanner_ack_mask := 0;
  scan1_trig := 32766; scan1_serial := reset_nonce;
  scan2_trig := 32766; scan2_serial := reset_nonce;
  scan3_trig := 32766; scan3_serial := reset_nonce;
  jam_alarm := FALSE; coll_alarm := FALSE;
  noread_alarm := FALSE; nohome_alarm := FALSE;
  auto_mode := TRUE;
  lane1_run := TRUE; lane2_run := TRUE; lane3_run := TRUE;
  ob1_run := TRUE; ob2_run := TRUE; ob3_run := TRUE;
  init_done := TRUE;
END_IF;

(* logical clock. Wraps at INT max; a run is not expected to reach it,
   and a wrap is visible as a discontinuity rather than silently wrong. *)
IF scan_ct < 32000 THEN
  scan_ct := scan_ct + 1;
ELSE
  scan_ct := 0;
END_IF;

(* XLe must provision a journal-backed identity while stopped. A stale offer
   present at PLC startup is ignored until its commit ID changes. *)
IF epoch_offer_id <> 0 AND epoch_offer_id <> epoch_offer_seen THEN
  epoch_offer_seen := epoch_offer_id;
  epoch_ack_id := epoch_offer_id;
  IF NOT sorter_run AND scanner_state = 0 AND
     epoch_active_lo = 0 AND epoch_active_hi = 0 AND
     epoch_offer_lo >= 0 AND epoch_offer_lo < 30000 AND
     epoch_offer_hi >= 0 AND epoch_offer_hi < 30000 AND
     (epoch_offer_lo <> 0 OR epoch_offer_hi <> 0) THEN
    epoch_active_lo := epoch_offer_lo; epoch_active_hi := epoch_offer_hi;
    hb_seen := hb_sequence; hb_age := 0; hb_ready := FALSE;
  END_IF;
END_IF;
IF epoch_fault_request = 2 THEN
  epoch_fault := 2;
ELSIF epoch_active_lo = 0 AND epoch_active_hi = 0 THEN
  epoch_fault := 1;
ELSE
  epoch_fault := 0;
END_IF;

(* A changed heartbeat is valid only for this journal-backed run. The PLC
   keeps belts moving on loss so accepted routes finish and undecided
   packages recirculate. Only induction and new route commands are held. *)
IF xle_mode AND xle_multi AND epoch_fault = 0 THEN
  IF hb_sequence <> 0 AND hb_sequence <> hb_seen THEN
    hb_seen := hb_sequence;
    IF hb_epoch_lo = epoch_active_lo AND hb_epoch_hi = epoch_active_hi THEN
      hb_age := 0; hb_ready := TRUE; hb_ack_sequence := hb_sequence;
    END_IF;
  END_IF;
  IF hb_age < 32000 THEN hb_age := hb_age + 1; END_IF;
  IF hb_age > 50 THEN
    hb_ready := FALSE;
    IF xle_liveness = 0 OR xle_liveness = 3 THEN
      xle_liveness := 1;
    END_IF;
  END_IF;
END_IF;
IF xle_liveness = 1 AND xle_fault_ack THEN
  xle_liveness := 2;
END_IF;
xle_fault_ack := FALSE;
IF xle_liveness = 2 AND xle_retry AND hb_ready AND hb_age <= 50 THEN
  recovery_seen := recovery_sequence;
  xle_liveness := 3;
END_IF;
xle_retry := FALSE;
IF xle_liveness = 3 AND hb_ready AND hb_age <= 50 AND
   recovery_sequence <> 0 AND recovery_sequence <> recovery_seen THEN
  recovery_seen := recovery_sequence;
  IF recovery_epoch_lo = epoch_active_lo AND
     recovery_epoch_hi = epoch_active_hi THEN
    xle_liveness := 0;
  END_IF;
END_IF;

(* operator fault reset: latch the request into a held countdown so the
   bit survives long enough for the drives to sample it *)
IF fault_reset THEN
  frst_tmr := 10;
  fault_reset := FALSE;
END_IF;
IF frst_tmr > 0 THEN
  frst_tmr := frst_tmr - 1;
END_IF;

(* belt load, published to each drive *)
  occ := 0;
  FOR i := 0 TO 19 DO
    IF ib1[i] <> 0 THEN occ := occ + 1; END_IF;
  END_FOR;
  induct1_load := occ;
  occ := 0;
  FOR i := 0 TO 19 DO
    IF ib2[i] <> 0 THEN occ := occ + 1; END_IF;
  END_FOR;
  induct2_load := occ;
  occ := 0;
  FOR i := 0 TO 19 DO
    IF ib3[i] <> 0 THEN occ := occ + 1; END_IF;
  END_FOR;
  induct3_load := occ;
  occ := 0;
  FOR i := 0 TO 19 DO
    IF ob1[i] <> 0 THEN occ := occ + 1; END_IF;
  END_FOR;
  outbnd1_load := occ;
  occ := 0;
  FOR i := 0 TO 19 DO
    IF ob2[i] <> 0 THEN occ := occ + 1; END_IF;
  END_FOR;
  outbnd2_load := occ;
  occ := 0;
  FOR i := 0 TO 19 DO
    IF ob3[i] <> 0 THEN occ := occ + 1; END_IF;
  END_FOR;
  outbnd3_load := occ;

(* drive commands. Bit 2 is the fault reset and is asserted in both
   branches: a faulted drive is not running, so a reset that only
   reaches it while running would never clear anything. *)
IF sorter_run AND lane1_run THEN
  IF frst_tmr > 0 THEN induct1_cmd := 7; ELSE induct1_cmd := 3; END_IF;
  induct1_ref := speed_sp_1;
ELSE
  IF frst_tmr > 0 THEN induct1_cmd := 4; ELSE induct1_cmd := 0; END_IF;
  induct1_ref := 0;
END_IF;
IF sorter_run AND lane2_run THEN
  IF frst_tmr > 0 THEN induct2_cmd := 7; ELSE induct2_cmd := 3; END_IF;
  induct2_ref := speed_sp_2;
ELSE
  IF frst_tmr > 0 THEN induct2_cmd := 4; ELSE induct2_cmd := 0; END_IF;
  induct2_ref := 0;
END_IF;
IF sorter_run AND lane3_run THEN
  IF frst_tmr > 0 THEN induct3_cmd := 7; ELSE induct3_cmd := 3; END_IF;
  induct3_ref := speed_sp_3;
ELSE
  IF frst_tmr > 0 THEN induct3_cmd := 4; ELSE induct3_cmd := 0; END_IF;
  induct3_ref := 0;
END_IF;
IF sorter_run AND ob1_run THEN
  IF frst_tmr > 0 THEN outbnd1_cmd := 7; ELSE outbnd1_cmd := 3; END_IF;
  outbnd1_ref := ob_speed_1;
ELSE
  IF frst_tmr > 0 THEN outbnd1_cmd := 4; ELSE outbnd1_cmd := 0; END_IF;
  outbnd1_ref := 0;
END_IF;
IF sorter_run AND ob2_run THEN
  IF frst_tmr > 0 THEN outbnd2_cmd := 7; ELSE outbnd2_cmd := 3; END_IF;
  outbnd2_ref := ob_speed_2;
ELSE
  IF frst_tmr > 0 THEN outbnd2_cmd := 4; ELSE outbnd2_cmd := 0; END_IF;
  outbnd2_ref := 0;
END_IF;
IF sorter_run AND ob3_run THEN
  IF frst_tmr > 0 THEN outbnd3_cmd := 7; ELSE outbnd3_cmd := 3; END_IF;
  outbnd3_ref := ob_speed_3;
ELSE
  IF frst_tmr > 0 THEN outbnd3_cmd := 4; ELSE outbnd3_cmd := 0; END_IF;
  outbnd3_ref := 0;
END_IF;

(* ---------- camera tunnels ---------- *)
scan1_seed := master_seed; scan2_seed := master_seed; scan3_seed := master_seed;
scan1_nrrate := noread_sp; scan2_nrrate := noread_sp; scan3_nrrate := noread_sp;
IF scanner_state = 1 OR scanner_state = 2 THEN
  scanner_ack_mask := 0;
  IF scanner_state = 1 THEN
    IF scan1_result = 32766 AND scan1_status = 7 AND scan1_nonce = reset_nonce THEN scanner_ack_mask := scanner_ack_mask + 1; END_IF;
    IF scan2_result = 32766 AND scan2_status = 7 AND scan2_nonce = reset_nonce THEN scanner_ack_mask := scanner_ack_mask + 2; END_IF;
    IF scan3_result = 32766 AND scan3_status = 7 AND scan3_nonce = reset_nonce THEN scanner_ack_mask := scanner_ack_mask + 4; END_IF;
  ELSE
    IF scan1_result = 32767 AND scan1_status = 6 AND scan1_nonce = reset_nonce THEN scanner_ack_mask := scanner_ack_mask + 1; END_IF;
    IF scan2_result = 32767 AND scan2_status = 6 AND scan2_nonce = reset_nonce THEN scanner_ack_mask := scanner_ack_mask + 2; END_IF;
    IF scan3_result = 32767 AND scan3_status = 6 AND scan3_nonce = reset_nonce THEN scanner_ack_mask := scanner_ack_mask + 4; END_IF;
  END_IF;
  IF scanner_ack_mask = 7 THEN
    scanner_wait := 0;
    IF scanner_state = 1 THEN
      scanner_state := 2;
      scan1_trig := 32767; scan2_trig := 32767; scan3_trig := 32767;
    ELSE
      scanner_state := 0; scanner_fault_mask := 0;
      scan1_trig := 0; scan2_trig := 0; scan3_trig := 0;
    END_IF;
  ELSE
    scanner_wait := scanner_wait + 1;
    IF scanner_wait >= 200 THEN
      scanner_fault_mask := 7 - scanner_ack_mask;
      scanner_state := 3;
      sorter_run := FALSE;
    END_IF;
  END_IF;
ELSIF scanner_state = 3 THEN
  sorter_run := FALSE;
  IF scanner_fault_ack THEN scanner_state := 4; END_IF;
ELSIF scanner_state = 4 THEN
  sorter_run := FALSE;
  IF scanner_retry THEN
    reset_nonce := reset_nonce + 1;
    IF reset_nonce > 30000 THEN reset_nonce := 1; END_IF;
    xle_run_nonce := reset_nonce;
    scanner_state := 1; scanner_wait := 0; scanner_ack_mask := 0;
    scan1_trig := 32766; scan1_serial := reset_nonce;
    scan2_trig := 32766; scan2_serial := reset_nonce;
    scan3_trig := 32766; scan3_serial := reset_nonce;
  END_IF;
ELSE
(* tunnel 1: request a read on arrival, apply the answer when
   it comes back. Identity crosses a network hop and takes time, so
   a package can leave before its result arrives. That is a late
   scan, which is not the same thing as a failed read. *)
scan1_seed := master_seed;
scan1_nrrate := noread_sp;
IF NOT plant_mode THEN
IF ib1[10] = 0 OR ib1[10] <> tun_pkg_1 THEN
  IF tun_wait_1 THEN
    scan_late_ct := scan_late_ct + 1;
    tun_wait_1 := FALSE;
  END_IF;
  tun_pkg_1 := ib1[10];
  IF ib1[10] <> 0 THEN
    tun_seq_1 := tun_seq_1 + 1;
    IF tun_seq_1 > 30000 THEN tun_seq_1 := 1; END_IF;
    scan1_trig := tun_seq_1;
    scan1_serial := ib1[10];
    tun_wait_1 := TRUE;
  END_IF;
ELSIF tun_wait_1 AND scan1_result = tun_seq_1 AND scan1_nonce = reset_nonce THEN
  tun_wait_1 := FALSE;
  bc := scan1_bc;
  sts := scan1_status;
  scan_code_1 := bc;
  IF xle_mode AND xle_multi THEN
    FOR j := 0 TO 2 DO
      IF st_state[j] = 1 AND st_token[j] = tok1[10] THEN
        st_seq[j] := tun_seq_1;
        st_bc[j] := bc;
        st_scan[j] := scan_ct;
        st_state[j] := 2;
      END_IF;
    END_FOR;
  END_IF;
  IF sts = 0 OR sts = 3 OR sts = 4 THEN
    IF sts = 3 THEN oversize_ct := oversize_ct + 1; END_IF;
    IF sts = 4 THEN duplicate_ct := duplicate_ct + 1; END_IF;
    (* the package becomes what the tunnel says it is. Truth and
       belief part company here: the door scan compares this against
       the trailer it actually ends up in. *)
    ib1[10] := bc;
    tun_pkg_1 := bc;
    IF xle_mode THEN
      xle_package := bc;
      xle_state := 0; xle_reason := 0; xle_actual := 0;
      xle_route_dest := 0;
      xle_scan_tick := scan_ct;
      xle_accept_tick := 0; xle_divert_tick := 0;
      rt1[10] := 0;
    ELSE
      dest  := bc / 1000;
      obelt := ((dest - 1) / 3) + 1;
      IF obelt = 1 THEN rt1[10] := 14;
      ELSIF obelt = 2 THEN rt1[10] := 16;
      ELSIF obelt = 3 THEN rt1[10] := 18;
      ELSE rt1[10] := 0;
      END_IF;
    END_IF;
  ELSE
    (* no usable identity: the package keeps its serial, rides to the
       end of the belt and recirculates. *)
    rt1[10] := 0;
    IF sts = 1 THEN
      noread_ct := noread_ct + 1;
      noread_alarm := TRUE;
    ELSIF sts = 2 THEN
      multiple_ct := multiple_ct + 1;
    ELSIF sts = 5 THEN
      invalid_ct := invalid_ct + 1;
    END_IF;
  END_IF;
END_IF;
ELSE
  (* The tunnel photoeye, below, starts this request. The response is bound
     to its slot token, never to a barcode or a PLC belt cell. *)
  IF tun_wait_1 AND scan1_result = tun_seq_1 AND scan1_nonce = reset_nonce THEN
    tun_wait_1 := FALSE;
    scan_code_1 := scan1_bc;
    FOR j := 0 TO 2 DO
      IF st_state[j] = 1 AND st_lane[j] = 1 AND st_token[j] = plant_scan_token THEN
        st_seq[j] := tun_seq_1;
        st_bc[j] := scan1_bc;
        st_scan[j] := scan_ct;
        st_state[j] := 2;
        IF scan1_status = 1 THEN noread_ct := noread_ct + 1; noread_alarm := TRUE; END_IF;
        IF scan1_status = 2 THEN multiple_ct := multiple_ct + 1; END_IF;
        IF scan1_status = 3 THEN oversize_ct := oversize_ct + 1; END_IF;
        IF scan1_status = 4 THEN duplicate_ct := duplicate_ct + 1; END_IF;
        IF scan1_status = 5 THEN invalid_ct := invalid_ct + 1; END_IF;
      END_IF;
    END_FOR;
  END_IF;
END_IF;

(* tunnel 2: request a read on arrival, apply the answer when
   it comes back. Identity crosses a network hop and takes time, so
   a package can leave before its result arrives. That is a late
   scan, which is not the same thing as a failed read. *)
scan2_seed := master_seed;
scan2_nrrate := noread_sp;
IF NOT plant_mode THEN
IF ib2[10] = 0 OR ib2[10] <> tun_pkg_2 THEN
  IF tun_wait_2 THEN
    scan_late_ct := scan_late_ct + 1;
    tun_wait_2 := FALSE;
  END_IF;
  tun_pkg_2 := ib2[10];
  IF ib2[10] <> 0 THEN
    tun_seq_2 := tun_seq_2 + 1;
    IF tun_seq_2 > 30000 THEN tun_seq_2 := 1; END_IF;
    scan2_trig := tun_seq_2;
    scan2_serial := ib2[10];
    tun_wait_2 := TRUE;
  END_IF;
ELSIF tun_wait_2 AND scan2_result = tun_seq_2 AND scan2_nonce = reset_nonce THEN
  tun_wait_2 := FALSE;
  bc := scan2_bc;
  sts := scan2_status;
  scan_code_2 := bc;
  IF sts = 0 OR sts = 3 OR sts = 4 THEN
    IF sts = 3 THEN oversize_ct := oversize_ct + 1; END_IF;
    IF sts = 4 THEN duplicate_ct := duplicate_ct + 1; END_IF;
    (* the package becomes what the tunnel says it is. Truth and
       belief part company here: the door scan compares this against
       the trailer it actually ends up in. *)
    ib2[10] := bc;
    tun_pkg_2 := bc;
    dest  := bc / 1000;
    obelt := ((dest - 1) / 3) + 1;
    IF obelt = 1 THEN rt2[10] := 14;
    ELSIF obelt = 2 THEN rt2[10] := 16;
    ELSIF obelt = 3 THEN rt2[10] := 18;
    ELSE rt2[10] := 0;
    END_IF;
  ELSE
    (* no usable identity: the package keeps its serial, rides to the
       end of the belt and recirculates. *)
    rt2[10] := 0;
    IF sts = 1 THEN
      noread_ct := noread_ct + 1;
      noread_alarm := TRUE;
    ELSIF sts = 2 THEN
      multiple_ct := multiple_ct + 1;
    ELSIF sts = 5 THEN
      invalid_ct := invalid_ct + 1;
    END_IF;
  END_IF;
END_IF;
ELSE
  IF tun_wait_2 AND scan2_result = tun_seq_2 AND scan2_nonce = reset_nonce THEN
    tun_wait_2 := FALSE;
    scan_code_2 := scan2_bc;
    FOR j := 0 TO 2 DO
      IF st_state[j] = 1 AND st_lane[j] = 2 AND
         st_token[j] = plant_scan_token_2 THEN
        st_seq[j] := tun_seq_2;
        st_bc[j] := scan2_bc;
        st_scan[j] := scan_ct;
        st_state[j] := 2;
        IF scan2_status = 1 THEN noread_ct := noread_ct + 1; noread_alarm := TRUE; END_IF;
        IF scan2_status = 2 THEN multiple_ct := multiple_ct + 1; END_IF;
        IF scan2_status = 3 THEN oversize_ct := oversize_ct + 1; END_IF;
        IF scan2_status = 4 THEN duplicate_ct := duplicate_ct + 1; END_IF;
        IF scan2_status = 5 THEN invalid_ct := invalid_ct + 1; END_IF;
      END_IF;
    END_FOR;
  END_IF;
END_IF;

(* tunnel 3: request a read on arrival, apply the answer when
   it comes back. Identity crosses a network hop and takes time, so
   a package can leave before its result arrives. That is a late
   scan, which is not the same thing as a failed read. *)
scan3_seed := master_seed;
scan3_nrrate := noread_sp;
IF NOT plant_mode THEN
IF ib3[10] = 0 OR ib3[10] <> tun_pkg_3 THEN
  IF tun_wait_3 THEN
    scan_late_ct := scan_late_ct + 1;
    tun_wait_3 := FALSE;
  END_IF;
  tun_pkg_3 := ib3[10];
  IF ib3[10] <> 0 THEN
    tun_seq_3 := tun_seq_3 + 1;
    IF tun_seq_3 > 30000 THEN tun_seq_3 := 1; END_IF;
    scan3_trig := tun_seq_3;
    scan3_serial := ib3[10];
    tun_wait_3 := TRUE;
  END_IF;
ELSIF tun_wait_3 AND scan3_result = tun_seq_3 AND scan3_nonce = reset_nonce THEN
  tun_wait_3 := FALSE;
  bc := scan3_bc;
  sts := scan3_status;
  scan_code_3 := bc;
  IF sts = 0 OR sts = 3 OR sts = 4 THEN
    IF sts = 3 THEN oversize_ct := oversize_ct + 1; END_IF;
    IF sts = 4 THEN duplicate_ct := duplicate_ct + 1; END_IF;
    (* the package becomes what the tunnel says it is. Truth and
       belief part company here: the door scan compares this against
       the trailer it actually ends up in. *)
    ib3[10] := bc;
    tun_pkg_3 := bc;
    dest  := bc / 1000;
    obelt := ((dest - 1) / 3) + 1;
    IF obelt = 1 THEN rt3[10] := 14;
    ELSIF obelt = 2 THEN rt3[10] := 16;
    ELSIF obelt = 3 THEN rt3[10] := 18;
    ELSE rt3[10] := 0;
    END_IF;
  ELSE
    (* no usable identity: the package keeps its serial, rides to the
       end of the belt and recirculates. *)
    rt3[10] := 0;
    IF sts = 1 THEN
      noread_ct := noread_ct + 1;
      noread_alarm := TRUE;
    ELSIF sts = 2 THEN
      multiple_ct := multiple_ct + 1;
    ELSIF sts = 5 THEN
      invalid_ct := invalid_ct + 1;
    END_IF;
  END_IF;
END_IF;
ELSE
  IF tun_wait_3 AND scan3_result = tun_seq_3 AND scan3_nonce = reset_nonce THEN
    tun_wait_3 := FALSE;
    scan_code_3 := scan3_bc;
    FOR j := 0 TO 2 DO
      IF st_state[j] = 1 AND st_lane[j] = 3 AND
         st_token[j] = plant_scan_token_3 THEN
        st_seq[j] := tun_seq_3;
        st_bc[j] := scan3_bc;
        st_scan[j] := scan_ct;
        st_state[j] := 2;
        IF scan3_status = 1 THEN noread_ct := noread_ct + 1; noread_alarm := TRUE; END_IF;
        IF scan3_status = 2 THEN multiple_ct := multiple_ct + 1; END_IF;
        IF scan3_status = 3 THEN oversize_ct := oversize_ct + 1; END_IF;
        IF scan3_status = 4 THEN duplicate_ct := duplicate_ct + 1; END_IF;
        IF scan3_status = 5 THEN invalid_ct := invalid_ct + 1; END_IF;
      END_IF;
    END_FOR;
  END_IF;
END_IF;

(* Selected chute switch is independent of cumulative trailer counters. The
   plant commits a versioned raw sample; only this validator publishes state. *)
IF chute_mode THEN
  chute_permissive := 0;
  IF chute_resume_grace > 0 THEN
    chute_resume_grace := chute_resume_grace - 1;
  END_IF;
  IF NOT plant_mode OR NOT photoeye_mode OR NOT accumulation_mode OR
     chute_config_trailer <> 2 OR chute_config_capacity <> 3 THEN
    chute_quality := 3; chute_state := 4; sorter_run := FALSE;
  ELSE
    IF chute_raw_commit <> 0 AND chute_raw_commit = chute_raw_seq AND
       chute_raw_commit <> chute_seen THEN
      chute_expect := chute_seen + 1;
      IF chute_expect > 30000 THEN chute_expect := 1; END_IF;
      chute_identity_ok := chute_raw_token = 0 AND chute_raw_serial = 0 AND
                           chute_raw_reserved = 0;
      IF chute_raw_token <> 0 AND chute_raw_serial <> 0 THEN
        FOR j := 0 TO 2 DO
          IF st_token[j] = chute_raw_token AND st_serial[j] = chute_raw_serial AND
             st_lane[j] >= 1 AND st_lane[j] <= 3 THEN
            chute_identity_ok := TRUE;
          END_IF;
        END_FOR;
        IF chute_raw_token = chute_accepted_token AND
           chute_raw_serial = chute_accepted_serial THEN
          chute_identity_ok := TRUE;
        END_IF;
      END_IF;
      chute_valid := chute_raw_version = 1 AND chute_raw_trailer = 2 AND
        chute_raw_epoch_lo = epoch_active_lo AND
        chute_raw_epoch_hi = epoch_active_hi AND
        chute_raw_nonce = reset_nonce AND chute_raw_seq = chute_expect AND
        chute_raw_occupied >= 0 AND chute_raw_occupied <= 3 AND
        chute_raw_reserved >= 0 AND chute_raw_reserved <= 3 AND
        chute_raw_occupied + chute_raw_reserved <= 3 AND
        chute_raw_full >= 0 AND chute_raw_full <= 1 AND
        ((chute_raw_occupied + chute_raw_reserved >= 3 AND
          chute_raw_full = 1) OR
         (chute_raw_occupied + chute_raw_reserved < 3 AND
          chute_raw_full = 0)) AND chute_identity_ok;
      IF chute_raw_occupied > chute_view_occupied THEN
        chute_valid := chute_valid AND
          chute_raw_occupied = chute_view_occupied + 1 AND
          chute_raw_accepted_token = chute_accepted_token AND
          chute_raw_accepted_serial = chute_accepted_serial AND
          chute_raw_accepted_seq = chute_accepted_event_seq AND
          chute_raw_accepted_seq <> 0 AND
          (chute_raw_accepted_token <> chute_accounted_token OR
           chute_raw_accepted_serial <> chute_accounted_serial OR
           chute_raw_accepted_seq <> chute_accounted_seq);
      END_IF;
      IF chute_raw_occupied < chute_view_occupied THEN
        chute_valid := chute_valid AND chute_empty_ack = chute_empty_seq AND
          chute_empty_result = 1 AND chute_empty_seq <> 0 AND
          chute_raw_occupied = 0 AND chute_raw_reserved = 0;
      END_IF;
      chute_seen := chute_raw_seq;
      IF chute_valid THEN
        chute_raw_ack := chute_seen; chute_quality := 1; chute_age := 0;
        IF chute_raw_occupied > chute_view_occupied THEN
          chute_accounted_token := chute_raw_accepted_token;
          chute_accounted_serial := chute_raw_accepted_serial;
          chute_accounted_seq := chute_raw_accepted_seq;
        END_IF;
        chute_view_trailer := 2; chute_view_occupied := chute_raw_occupied;
        IF chute_raw_full = 1 THEN
          IF chute_state <> 2 THEN chute_state := 1; END_IF;
        ELSIF chute_state = 1 OR chute_state = 2 THEN
          IF chute_empty_ack = chute_empty_seq AND chute_empty_result = 1 AND
             chute_empty_seq <> 0 THEN
            chute_state := 3;
          ELSE
            chute_quality := 3; chute_state := 4; sorter_run := FALSE;
          END_IF;
        END_IF;
      ELSE
        chute_quality := 3; chute_state := 4; sorter_run := FALSE;
      END_IF;
    ELSIF chute_age < 32000 THEN
      chute_age := chute_age + 1;
    END_IF;
    IF chute_age > 15 THEN
      chute_quality := 2; chute_state := 4; sorter_run := FALSE;
    END_IF;
    IF chute_action_seq <> 0 AND chute_action_seq <> chute_action_seen THEN
      chute_action_expect := chute_action_seen + 1;
      IF chute_action_expect > 30000 THEN chute_action_expect := 1; END_IF;
      chute_action_seen := chute_action_seq;
      chute_action_ack := chute_action_seq;
      chute_action_result := 3;
      IF chute_action_seq = chute_action_expect AND
         chute_action_trailer = 2 AND
         chute_action_epoch_lo = epoch_active_lo AND
         chute_action_epoch_hi = epoch_active_hi AND
         chute_action_nonce = reset_nonce AND chute_quality = 1 THEN
        chute_action_result := 2;
        IF chute_action_op = 1 AND chute_state = 1 THEN
          chute_state := 2; chute_action_result := 1;
        ELSIF chute_action_op = 2 AND chute_state = 2 AND
              chute_raw_reserved = 0 AND chute_view_occupied = 3 THEN
          chute_empty_next := chute_empty_next + 1;
          IF chute_empty_next > 30000 THEN chute_empty_next := 1; END_IF;
          chute_empty_trailer := 2;
          chute_empty_epoch_lo := epoch_active_lo;
          chute_empty_epoch_hi := epoch_active_hi;
          chute_empty_nonce := reset_nonce;
          chute_empty_result := 0;
          chute_empty_seq := chute_empty_next;
          chute_action_result := 1;
        ELSIF chute_action_op = 3 AND chute_state = 3 AND
              chute_raw_occupied = 0 AND chute_raw_reserved = 0 AND
              chute_raw_full = 0 AND chute_empty_ack = chute_empty_seq AND
              chute_empty_result = 1 AND plant_fault = 0 AND z_fault = 0 AND
              pe_fault_mask = 0 AND epoch_fault = 0 AND xle_liveness = 0 THEN
          chute_state := 0; chute_action_result := 1;
          chute_resume_grace := 15;
        END_IF;
      END_IF;
    END_IF;
    IF chute_quality = 1 AND chute_state = 0 THEN
      chute_permissive := 1;
    END_IF;
  END_IF;
ELSE
  chute_state := 0; chute_quality := 0; chute_age := 0;
  chute_view_trailer := 0; chute_view_occupied := 0;
  chute_permissive := 1;
  chute_resume_grace := 0;
END_IF;

(* A plant commit is a seqlock over all three zone rows. Only the PLC may
   publish these bounded states. The rows cannot create route or outcome. *)
IF plant_mode AND accumulation_mode THEN
  z_raw_zone[0] := z0_raw_zone; z_raw_motion[0] := z0_raw_motion;
  z_raw_hold[0] := z0_raw_hold; z_raw_dwell[0] := z0_raw_dwell;
  z_raw_seq[0] := z0_raw_seq;
  z_raw_zone[1] := z1_raw_zone; z_raw_motion[1] := z1_raw_motion;
  z_raw_hold[1] := z1_raw_hold; z_raw_dwell[1] := z1_raw_dwell;
  z_raw_seq[1] := z1_raw_seq;
  z_raw_zone[2] := z2_raw_zone; z_raw_motion[2] := z2_raw_motion;
  z_raw_hold[2] := z2_raw_hold; z_raw_dwell[2] := z2_raw_dwell;
  z_raw_seq[2] := z2_raw_seq;
  z_belt[0] := p0_raw_belt; z_pos[0] := p0_raw_pos;
  z_belt[1] := p1_raw_belt; z_pos[1] := p1_raw_pos;
  z_belt[2] := p2_raw_belt; z_pos[2] := p2_raw_pos;
  IF z_raw_commit <> 0 AND z_raw_commit <> z_seen_commit THEN
    z_seen_commit := z_raw_commit;
    z_view_age := 0;
    IF z_raw_ready >= 0 AND z_raw_ready <= 7 AND
       plant_epoch_lo = epoch_active_lo AND plant_epoch_hi = epoch_active_hi AND
       plant_nonce = reset_nonce THEN
      z_view_ready := z_raw_ready;
    ELSE
      z_view_ready := 0; z_fault := 1;
    END_IF;
    FOR j := 0 TO 2 DO
      IF st_state[j] = 0 OR st_token[j] = 0 THEN
        z_quality[j] := 0; z_bound_token[j] := 0;
        z_view_zone[j] := 0; z_view_motion[j] := 0;
        z_view_hold[j] := 0; z_view_dwell[j] := 0;
      ELSIF z_bound_token[j] <> st_token[j] THEN
        (* A new PLC slot may appear after the plant read this cycle. Bind
           first and wait for the next complete plant commit. *)
        z_bound_token[j] := st_token[j]; z_view_zone[j] := 0;
        z_view_seq[j] := 0; z_quality[j] := 0;
      ELSIF st_state[j] = 1 AND z_raw_zone[j] = 0 THEN
        z_quality[j] := 0;
      ELSIF st_state[j] >= 5 AND z_raw_zone[j] = 0 THEN
        (* The plant's short terminal-history cache may expire before XLe
           releases a PLC slot. Keep the last validated coordinate stale. *)
        z_quality[j] := 2;
      ELSE
        z_valid := z_raw_seq[j] <> 0 AND z_raw_seq[j] <> z_view_seq[j] AND
          z_raw_zone[j] >= 1 AND z_raw_zone[j] <= 7 AND
          z_raw_motion[j] >= 1 AND z_raw_motion[j] <= 7 AND
          z_raw_hold[j] >= 0 AND z_raw_hold[j] <= 5 AND
          (z_raw_hold[j] <> 5 OR
          (chute_mode AND chute_permissive = 0 AND
            st_dest[j] = 2 AND
            (z_raw_motion[j] = 2 OR z_raw_motion[j] = 3)) OR
           (chute_mode AND chute_resume_grace > 0 AND
            st_dest[j] = 2 AND z_view_hold[j] = 5 AND
            z_view_zone[j] = z_raw_zone[j] AND
            z_view_motion[j] = z_raw_motion[j] AND
            (z_raw_motion[j] = 2 OR z_raw_motion[j] = 3))) AND
          z_raw_dwell[j] >= 0 AND z_raw_dwell[j] <= 32000 AND
          z_pos[j] >= 0 AND z_pos[j] <= 300;
        IF j = 0 THEN
          z_valid := z_valid AND z_raw_seq[j] = p0_raw_seq AND
            p0_raw_epoch_lo = epoch_active_lo AND p0_raw_epoch_hi = epoch_active_hi AND
            p0_raw_nonce = reset_nonce AND p0_raw_token = st_token[j] AND
            p0_raw_serial = st_serial[j];
        ELSIF j = 1 THEN
          z_valid := z_valid AND z_raw_seq[j] = p1_raw_seq AND
            p1_raw_epoch_lo = epoch_active_lo AND p1_raw_epoch_hi = epoch_active_hi AND
            p1_raw_nonce = reset_nonce AND p1_raw_token = st_token[j] AND
            p1_raw_serial = st_serial[j];
        ELSE
          z_valid := z_valid AND z_raw_seq[j] = p2_raw_seq AND
            p2_raw_epoch_lo = epoch_active_lo AND p2_raw_epoch_hi = epoch_active_hi AND
            p2_raw_nonce = reset_nonce AND p2_raw_token = st_token[j] AND
            p2_raw_serial = st_serial[j];
        END_IF;
        IF NOT z_valid THEN
          z_quality[j] := 3; z_fault := 1;
        ELSE
          IF (z_view_zone[j] <> 0 AND
              (z_raw_zone[j] < z_view_zone[j] OR
               z_raw_zone[j] > z_view_zone[j] + 1 AND
               NOT (z_view_zone[j] = 3 AND z_raw_zone[j] = 5) AND
               (* Zone 7 is the bounded lane recirculation tail. A route
                  decision may never enter it; the plant fixes fallback at 14. *)
               NOT (z_view_zone[j] = 3 AND z_raw_zone[j] = 7 AND
                    st_dest[j] = 0 AND (st_state[j] = 2 OR st_state[j] = 4 OR
                                       st_state[j] = 6)))) OR
             (z_raw_zone[j] = 1 AND z_pos[j] > 95) OR
             (z_raw_zone[j] = 2 AND (z_pos[j] < 85 OR z_pos[j] > 123)) OR
             (z_raw_zone[j] = 3 AND (z_pos[j] < 113 OR z_pos[j] >= 140)) OR
             (z_raw_zone[j] = 4 AND (z_pos[j] < 130 OR z_pos[j] > 140)) OR
             (z_raw_zone[j] = 5 AND (z_belt[j] < 2 OR z_belt[j] > 4)) OR
             (z_raw_zone[j] = 7 AND
              (z_pos[j] < 140 OR z_pos[j] > 190 OR st_dest[j] <> 0 OR
               NOT (st_state[j] = 2 OR st_state[j] = 4 OR st_state[j] = 6))) OR
             ((z_raw_zone[j] <= 4 OR z_raw_zone[j] = 7) AND
              NOT ((st_lane[j] = 1 AND z_belt[j] = 1) OR
                   (st_lane[j] = 2 AND z_belt[j] = 5) OR
                   (st_lane[j] = 3 AND z_belt[j] = 6))) THEN
            z_quality[j] := 3; z_fault := 2;
          ELSE
            z_view_zone[j] := z_raw_zone[j];
            z_view_motion[j] := z_raw_motion[j];
            z_view_hold[j] := z_raw_hold[j];
            z_view_dwell[j] := z_raw_dwell[j];
            z_view_seq[j] := z_raw_seq[j]; z_quality[j] := 1;
          END_IF;
        END_IF;
      END_IF;
    END_FOR;
    FOR j := 0 TO 2 DO
      IF z_quality[j] = 1 AND (z_view_zone[j] < 6 OR z_view_zone[j] = 7) THEN
        FOR i := j + 1 TO 2 DO
          IF z_quality[i] = 1 AND (z_view_zone[i] < 6 OR z_view_zone[i] = 7) AND
             z_belt[j] = z_belt[i] THEN
            z_difference := z_pos[j] - z_pos[i];
            IF z_difference < 0 THEN z_difference := -z_difference; END_IF;
            IF z_difference < 32 THEN
              z_quality[j] := 3; z_quality[i] := 3; z_fault := 3;
            END_IF;
          END_IF;
        END_FOR;
      END_IF;
    END_FOR;
  ELSIF z_view_age < 32000 THEN
    z_view_age := z_view_age + 1;
  END_IF;
  IF z_view_age > 15 THEN
    z_view_ready := 0;
    FOR j := 0 TO 2 DO
      IF z_quality[j] = 1 THEN z_quality[j] := 2; END_IF;
    END_FOR;
  END_IF;
  IF z_fault <> 0 THEN sorter_run := FALSE; z_view_ready := 0; END_IF;
  z0_view_zone := z_view_zone[0]; z0_view_motion := z_view_motion[0];
  z0_view_hold := z_view_hold[0]; z0_view_dwell := z_view_dwell[0];
  z0_view_seq := z_view_seq[0]; z0_quality := z_quality[0];
  z1_view_zone := z_view_zone[1]; z1_view_motion := z_view_motion[1];
  z1_view_hold := z_view_hold[1]; z1_view_dwell := z_view_dwell[1];
  z1_view_seq := z_view_seq[1]; z1_quality := z_quality[1];
  z2_view_zone := z_view_zone[2]; z2_view_motion := z_view_motion[2];
  z2_view_hold := z_view_hold[2]; z2_view_dwell := z_view_dwell[2];
  z2_view_seq := z_view_seq[2]; z2_quality := z_quality[2];
END_IF;

(* Opt-in stateful field inputs. The plant publishes three committed rows,
   one for each PLC slot. Only an exact run/lane/token/serial match is
   conditioned and copied to the supervisory view. Faults latch to reset. *)
IF plant_mode AND photoeye_mode THEN
  pe_epoch_lo[0] := pe0_raw_epoch_lo; pe_epoch_hi[0] := pe0_raw_epoch_hi;
  pe_nonce[0] := pe0_raw_nonce; pe_token[0] := pe0_raw_token;
  pe_serial[0] := pe0_raw_serial; pe_lane[0] := pe0_raw_lane;
  pe_mask[0] := pe0_raw_mask; pe_seq[0] := pe0_raw_seq;
  pe_epoch_lo[1] := pe1_raw_epoch_lo; pe_epoch_hi[1] := pe1_raw_epoch_hi;
  pe_nonce[1] := pe1_raw_nonce; pe_token[1] := pe1_raw_token;
  pe_serial[1] := pe1_raw_serial; pe_lane[1] := pe1_raw_lane;
  pe_mask[1] := pe1_raw_mask; pe_seq[1] := pe1_raw_seq;
  pe_epoch_lo[2] := pe2_raw_epoch_lo; pe_epoch_hi[2] := pe2_raw_epoch_hi;
  pe_nonce[2] := pe2_raw_nonce; pe_token[2] := pe2_raw_token;
  pe_serial[2] := pe2_raw_serial; pe_lane[2] := pe2_raw_lane;
  pe_mask[2] := pe2_raw_mask; pe_seq[2] := pe2_raw_seq;
  IF pe_debounce_sp >= 1 AND pe_debounce_sp <= 5 THEN
    pe_debounce := pe_debounce_sp;
  ELSE pe_debounce := 2; END_IF;
  IF pe_min_block_sp >= 1 AND pe_min_block_sp <= 30 THEN
    pe_min_block := pe_min_block_sp;
  ELSE pe_min_block := 2; END_IF;
  IF pe_max_block_sp >= 2 AND pe_max_block_sp <= 300 THEN
    pe_max_block := pe_max_block_sp;
  ELSE pe_max_block := 120; END_IF;
  IF pe_travel_sp >= 5 AND pe_travel_sp <= 1000 THEN
    pe_max_travel := pe_travel_sp;
  ELSE pe_max_travel := 400; END_IF;
  FOR j := 0 TO 2 DO
    IF st_state[j] = 0 OR st_token[j] = 0 THEN
      pe_bound_token[j] := 0; pe_seen[j] := pe_seq[j];
      pe_raw[j] := 0; pe_filtered[j] := 0; pe_age[j] := 0;
      pe_expected[j] := 1; pe_travel[j] := 0;
    ELSE
      IF pe_bound_token[j] <> st_token[j] THEN
        pe_bound_token[j] := st_token[j]; pe_seen[j] := pe_seq[j];
        pe_raw[j] := 0; pe_filtered[j] := 0; pe_age[j] := 0;
        pe_quality[j] := 0; pe_expected[j] := 1; pe_travel[j] := 0;
        FOR pe_sensor := 0 TO 4 DO
          pe_index := j * 5 + pe_sensor;
          pe_candidate[pe_index] := 0; pe_duration[pe_index] := 0;
          pe_stable[pe_index] := FALSE;
        END_FOR;
      END_IF;
      IF pe_seq[j] <> 0 AND pe_seq[j] <> pe_seen[j] THEN
        pe_seen[j] := pe_seq[j]; pe_age[j] := 0;
        IF pe_epoch_lo[j] = epoch_active_lo AND
           pe_epoch_hi[j] = epoch_active_hi AND
           pe_nonce[j] = reset_nonce AND pe_token[j] = st_token[j] AND
           pe_serial[j] = st_serial[j] AND pe_lane[j] = st_lane[j] AND
           pe_mask[j] >= 0 AND pe_mask[j] <= 31 THEN
          pe_raw[j] := pe_mask[j];
        ELSE
          pe_quality[j] := 1; pe_fault_sensor := pe_expected[j];
        END_IF;
      ELSIF pe_age[j] < 32000 THEN
        pe_age[j] := pe_age[j] + 1;
      END_IF;
      IF pe_age[j] > 15 AND pe_quality[j] = 0 THEN
        pe_quality[j] := 6; pe_fault_sensor := pe_expected[j];
      END_IF;
      IF pe_quality[j] = 0 AND pe_seen[j] <> 0 THEN
        pe_filtered[j] := 0;
        pe_bit := 1;
        FOR pe_sensor := 1 TO 5 DO
          pe_index := j * 5 + pe_sensor - 1;
          pe_is_raw := ((pe_raw[j] / pe_bit) MOD 2) = 1;
          IF pe_is_raw <> pe_stable[pe_index] THEN
            pe_candidate[pe_index] := pe_candidate[pe_index] + 1;
            IF pe_candidate[pe_index] >= pe_debounce THEN
              pe_candidate[pe_index] := 0;
              pe_stable[pe_index] := pe_is_raw;
              IF pe_is_raw THEN
                pe_duration[pe_index] := 0;
                IF pe_sensor <> pe_expected[j] THEN
                  (* Attribute a skipped transition to the beam that was
                     expected, rather than the downstream beam that exposed it. *)
                  pe_quality[j] := 5; pe_fault_sensor := pe_expected[j];
                ELSE
                  pe_travel[j] := 0;
                END_IF;
              ELSE
                IF pe_duration[pe_index] < pe_min_block THEN
                  pe_quality[j] := 4; pe_fault_sensor := pe_sensor;
                ELSIF pe_sensor = pe_expected[j] THEN
                  pe_expected[j] := pe_expected[j] + 1;
                  pe_travel[j] := 0;
                END_IF;
                pe_duration[pe_index] := 0;
              END_IF;
            END_IF;
          ELSE
            pe_candidate[pe_index] := 0;
          END_IF;
          IF pe_stable[pe_index] THEN
            pe_filtered[j] := pe_filtered[j] + pe_bit;
            IF accumulation_mode AND z_quality[j] = 1 AND
               (z_view_motion[j] = 2 OR z_view_motion[j] = 3 OR
                z_view_motion[j] = 4 OR z_view_motion[j] = 5) THEN
              (* The beam is physically blocked through a controlled hold.
                 A trailing edge must still satisfy the minimum duration. *)
              IF pe_duration[pe_index] < pe_min_block THEN
                pe_duration[pe_index] := pe_min_block;
              END_IF;
            ELSE
              IF pe_duration[pe_index] < 32000 THEN
                pe_duration[pe_index] := pe_duration[pe_index] + 1;
              END_IF;
              IF pe_duration[pe_index] > pe_max_block THEN
                pe_quality[j] := 3; pe_fault_sensor := pe_sensor;
              END_IF;
            END_IF;
          END_IF;
          pe_bit := pe_bit * 2;
        END_FOR;
        IF pe_expected[j] <= 5 AND pe_travel[j] < 32000 AND
           NOT (accumulation_mode AND z_quality[j] = 1 AND
                (z_view_motion[j] = 2 OR z_view_motion[j] = 3 OR
                 z_view_motion[j] = 4 OR z_view_motion[j] = 5)) THEN
          pe_travel[j] := pe_travel[j] + 1;
          IF pe_travel[j] > pe_max_travel THEN
            pe_quality[j] := 2; pe_fault_sensor := pe_expected[j];
          END_IF;
        END_IF;
      END_IF;
      IF pe_quality[j] <> 0 THEN
        IF j = 0 AND (pe_fault_mask MOD 2) = 0 THEN
          pe_fault_mask := pe_fault_mask + 1; END_IF;
        IF j = 1 AND ((pe_fault_mask / 2) MOD 2) = 0 THEN
          pe_fault_mask := pe_fault_mask + 2; END_IF;
        IF j = 2 AND ((pe_fault_mask / 4) MOD 2) = 0 THEN
          pe_fault_mask := pe_fault_mask + 4; END_IF;
        pe_fault_lane := st_lane[j]; sorter_run := FALSE;
      END_IF;
    END_IF;
  END_FOR;
  pe0_view_epoch_lo := epoch_active_lo; pe0_view_epoch_hi := epoch_active_hi;
  pe0_view_nonce := reset_nonce; pe0_view_token := pe_bound_token[0];
  pe0_view_serial := st_serial[0]; pe0_view_raw := pe_raw[0];
  pe0_view_conditioned := pe_filtered[0]; pe0_view_quality := pe_quality[0];
  pe1_view_epoch_lo := epoch_active_lo; pe1_view_epoch_hi := epoch_active_hi;
  pe1_view_nonce := reset_nonce; pe1_view_token := pe_bound_token[1];
  pe1_view_serial := st_serial[1]; pe1_view_raw := pe_raw[1];
  pe1_view_conditioned := pe_filtered[1]; pe1_view_quality := pe_quality[1];
  pe2_view_epoch_lo := epoch_active_lo; pe2_view_epoch_hi := epoch_active_hi;
  pe2_view_nonce := reset_nonce; pe2_view_token := pe_bound_token[2];
  pe2_view_serial := st_serial[2]; pe2_view_raw := pe_raw[2];
  pe2_view_conditioned := pe_filtered[2]; pe2_view_quality := pe_quality[2];
END_IF;

(* Plant events are serialized by the event/ack pair. The plant writes
   payload first and sequence last. The PLC accepts only its current run and
   an occupied slot with the exact token and serial. No counter advances on
   a route decision: only a physical confirmation can load a trailer. *)
IF plant_mode THEN
  l1_div1 := FALSE; l1_div2 := FALSE; l1_div3 := FALSE;
  l2_div1 := FALSE; l2_div2 := FALSE; l2_div3 := FALSE;
  l3_div1 := FALSE; l3_div2 := FALSE; l3_div3 := FALSE;
  IF plant_heartbeat <> plant_hb_seen THEN
    plant_hb_seen := plant_heartbeat; plant_hb_age := 0;
  ELSIF plant_hb_age < 32000 THEN
    plant_hb_age := plant_hb_age + 1;
  END_IF;
  IF plant_fault <> 3 THEN
    plant_fault := 0;
    IF plant_hb_age > 30 THEN plant_fault := 1; END_IF;
    IF plant_epoch_lo <> epoch_active_lo OR plant_epoch_hi <> epoch_active_hi OR
       plant_nonce <> reset_nonce THEN plant_fault := 2; END_IF;
    IF NOT xle_mode OR NOT xle_multi THEN plant_fault := 2; END_IF;
  END_IF;
  IF plant_fault <> 0 THEN sorter_run := FALSE; END_IF;
  (* Only identity-matched, bounded plant telemetry is published to SCADA.
     A stopped writer leaves its last coordinate intact but marks it stale. *)
  IF st_state[0] = 0 OR st_token[0] = 0 THEN
    p0_view_status := 0; p0_view_age := 0;
    p0_view_token := 0; p0_view_belt := 0;
    plant_view_seen0 := p0_raw_seq;
  ELSE
    IF p0_view_token <> 0 AND
       (p0_view_token <> st_token[0] OR p0_view_serial <> st_serial[0]) THEN
      p0_view_status := 3; p0_view_token := 0; p0_view_belt := 0;
      p0_view_age := 0;
    END_IF;
    IF p0_raw_seq <> 0 AND p0_raw_seq <> plant_view_seen0 THEN
      plant_view_seen0 := p0_raw_seq;
      IF p0_raw_epoch_lo = epoch_active_lo AND p0_raw_epoch_hi = epoch_active_hi AND
         p0_raw_nonce = reset_nonce AND p0_raw_token = st_token[0] AND
         p0_raw_serial = st_serial[0] AND
         ((st_lane[0] = 1 AND p0_raw_belt = 1) OR
          (st_lane[0] = 2 AND p0_raw_belt = 5) OR
          (st_lane[0] = 3 AND p0_raw_belt = 6) OR
          (p0_raw_belt >= 2 AND p0_raw_belt <= 4)) AND
         p0_raw_pos >= 0 AND p0_raw_pos <= 300 AND
         p0_raw_event >= 0 AND p0_raw_event <= 6 AND
         p0_raw_actual >= 0 AND p0_raw_actual <= 9 THEN
        p0_view_epoch_lo := p0_raw_epoch_lo; p0_view_epoch_hi := p0_raw_epoch_hi;
        p0_view_nonce := p0_raw_nonce; p0_view_token := p0_raw_token;
        p0_view_serial := p0_raw_serial; p0_view_belt := p0_raw_belt;
        p0_view_pos := p0_raw_pos; p0_view_event := p0_raw_event;
        p0_view_actual := p0_raw_actual; p0_view_seq := p0_raw_seq;
        p0_view_age := 0; p0_view_status := 1;
      ELSE
        p0_view_status := 3; p0_view_token := 0; p0_view_belt := 0;
      END_IF;
    ELSIF p0_view_age < 32000 THEN
      p0_view_age := p0_view_age + 1;
    END_IF;
    IF p0_view_age > 15 AND p0_view_status = 1 THEN p0_view_status := 2; END_IF;
  END_IF;
  IF st_state[1] = 0 OR st_token[1] = 0 THEN
    p1_view_status := 0; p1_view_age := 0;
    p1_view_token := 0; p1_view_belt := 0;
    plant_view_seen1 := p1_raw_seq;
  ELSE
    IF p1_view_token <> 0 AND
       (p1_view_token <> st_token[1] OR p1_view_serial <> st_serial[1]) THEN
      p1_view_status := 3; p1_view_token := 0; p1_view_belt := 0;
      p1_view_age := 0;
    END_IF;
    IF p1_raw_seq <> 0 AND p1_raw_seq <> plant_view_seen1 THEN
      plant_view_seen1 := p1_raw_seq;
      IF p1_raw_epoch_lo = epoch_active_lo AND p1_raw_epoch_hi = epoch_active_hi AND
         p1_raw_nonce = reset_nonce AND p1_raw_token = st_token[1] AND
         p1_raw_serial = st_serial[1] AND
         ((st_lane[1] = 1 AND p1_raw_belt = 1) OR
          (st_lane[1] = 2 AND p1_raw_belt = 5) OR
          (st_lane[1] = 3 AND p1_raw_belt = 6) OR
          (p1_raw_belt >= 2 AND p1_raw_belt <= 4)) AND
         p1_raw_pos >= 0 AND p1_raw_pos <= 300 AND
         p1_raw_event >= 0 AND p1_raw_event <= 6 AND
         p1_raw_actual >= 0 AND p1_raw_actual <= 9 THEN
        p1_view_epoch_lo := p1_raw_epoch_lo; p1_view_epoch_hi := p1_raw_epoch_hi;
        p1_view_nonce := p1_raw_nonce; p1_view_token := p1_raw_token;
        p1_view_serial := p1_raw_serial; p1_view_belt := p1_raw_belt;
        p1_view_pos := p1_raw_pos; p1_view_event := p1_raw_event;
        p1_view_actual := p1_raw_actual; p1_view_seq := p1_raw_seq;
        p1_view_age := 0; p1_view_status := 1;
      ELSE
        p1_view_status := 3; p1_view_token := 0; p1_view_belt := 0;
      END_IF;
    ELSIF p1_view_age < 32000 THEN
      p1_view_age := p1_view_age + 1;
    END_IF;
    IF p1_view_age > 15 AND p1_view_status = 1 THEN p1_view_status := 2; END_IF;
  END_IF;
  IF st_state[2] = 0 OR st_token[2] = 0 THEN
    p2_view_status := 0; p2_view_age := 0;
    p2_view_token := 0; p2_view_belt := 0;
    plant_view_seen2 := p2_raw_seq;
  ELSE
    IF p2_view_token <> 0 AND
       (p2_view_token <> st_token[2] OR p2_view_serial <> st_serial[2]) THEN
      p2_view_status := 3; p2_view_token := 0; p2_view_belt := 0;
      p2_view_age := 0;
    END_IF;
    IF p2_raw_seq <> 0 AND p2_raw_seq <> plant_view_seen2 THEN
      plant_view_seen2 := p2_raw_seq;
      IF p2_raw_epoch_lo = epoch_active_lo AND p2_raw_epoch_hi = epoch_active_hi AND
         p2_raw_nonce = reset_nonce AND p2_raw_token = st_token[2] AND
         p2_raw_serial = st_serial[2] AND
         ((st_lane[2] = 1 AND p2_raw_belt = 1) OR
          (st_lane[2] = 2 AND p2_raw_belt = 5) OR
          (st_lane[2] = 3 AND p2_raw_belt = 6) OR
          (p2_raw_belt >= 2 AND p2_raw_belt <= 4)) AND
         p2_raw_pos >= 0 AND p2_raw_pos <= 300 AND
         p2_raw_event >= 0 AND p2_raw_event <= 6 AND
         p2_raw_actual >= 0 AND p2_raw_actual <= 9 THEN
        p2_view_epoch_lo := p2_raw_epoch_lo; p2_view_epoch_hi := p2_raw_epoch_hi;
        p2_view_nonce := p2_raw_nonce; p2_view_token := p2_raw_token;
        p2_view_serial := p2_raw_serial; p2_view_belt := p2_raw_belt;
        p2_view_pos := p2_raw_pos; p2_view_event := p2_raw_event;
        p2_view_actual := p2_raw_actual; p2_view_seq := p2_raw_seq;
        p2_view_age := 0; p2_view_status := 1;
      ELSE
        p2_view_status := 3; p2_view_token := 0; p2_view_belt := 0;
      END_IF;
    ELSIF p2_view_age < 32000 THEN
      p2_view_age := p2_view_age + 1;
    END_IF;
    IF p2_view_age > 15 AND p2_view_status = 1 THEN p2_view_status := 2; END_IF;
  END_IF;
  pe_event_ready := TRUE;
  IF photoeye_mode AND plant_event_seq <> 0 AND plant_event_seq <> plant_seen THEN
    FOR j := 0 TO 2 DO
      IF st_token[j] = plant_event_token AND st_serial[j] = plant_event_serial AND
         st_lane[j] = plant_event_lane THEN
        IF pe_quality[j] <> 0 THEN pe_event_ready := FALSE; END_IF;
        IF plant_event_type = 1 AND pe_expected[j] < 2 THEN pe_event_ready := FALSE; END_IF;
        IF plant_event_type = 2 AND pe_expected[j] < 3 THEN pe_event_ready := FALSE; END_IF;
        IF plant_event_type = 3 AND pe_expected[j] < 4 THEN pe_event_ready := FALSE; END_IF;
        IF plant_event_type = 4 AND pe_expected[j] < 6 THEN pe_event_ready := FALSE; END_IF;
      END_IF;
    END_FOR;
  END_IF;
  IF plant_event_seq <> 0 AND plant_event_seq <> plant_seen AND pe_event_ready THEN
    plant_seen := plant_event_seq;
    plant_event_ack := plant_event_seq;
    slot_index := -1;
    plant_lane_match := FALSE;
    FOR j := 0 TO 2 DO
      IF st_state[j] <> 0 AND st_token[j] = plant_event_token AND
         st_serial[j] = plant_event_serial THEN
        slot_index := j;
        plant_lane_match := st_lane[j] = plant_event_lane;
      END_IF;
    END_FOR;
    IF plant_fault = 0 AND slot_index >= 0 AND plant_lane_match THEN
      j := slot_index;
      IF plant_event_type = 1 AND st_state[j] = 1 AND plant_request_pending THEN
        plant_request_pending := FALSE;
        inducted_ct := inducted_ct + 1;
      ELSIF plant_event_type = 2 AND st_state[j] = 1 THEN
        IF st_lane[j] = 1 THEN
          IF tun_wait_1 THEN scan_late_ct := scan_late_ct + 1; END_IF;
          tun_seq_1 := tun_seq_1 + 1;
          IF tun_seq_1 > 30000 THEN tun_seq_1 := 1; END_IF;
          scan1_trig := tun_seq_1;
          scan1_serial := st_serial[j];
          plant_scan_token := st_token[j];
          tun_wait_1 := TRUE;
        ELSIF st_lane[j] = 2 THEN
          IF tun_wait_2 THEN scan_late_ct := scan_late_ct + 1; END_IF;
          tun_seq_2 := tun_seq_2 + 1;
          IF tun_seq_2 > 30000 THEN tun_seq_2 := 1; END_IF;
          scan2_trig := tun_seq_2;
          scan2_serial := st_serial[j];
          plant_scan_token_2 := st_token[j];
          tun_wait_2 := TRUE;
        ELSIF st_lane[j] = 3 THEN
          IF tun_wait_3 THEN scan_late_ct := scan_late_ct + 1; END_IF;
          tun_seq_3 := tun_seq_3 + 1;
          IF tun_seq_3 > 30000 THEN tun_seq_3 := 1; END_IF;
          scan3_trig := tun_seq_3;
          scan3_serial := st_serial[j];
          plant_scan_token_3 := st_token[j];
          tun_wait_3 := TRUE;
        END_IF;
      ELSIF plant_event_type = 3 AND (st_state[j] = 2 OR st_state[j] = 3) THEN
        st_divert[j] := scan_ct;
        obelt := 0;
        IF st_dest[j] >= 1 AND st_dest[j] <= 9 THEN
          obelt := ((st_dest[j] - 1) / 3) + 1;
          IF obelt = 1 THEN
            IF st_lane[j] = 1 THEN l1_div1 := TRUE;
            ELSIF st_lane[j] = 2 THEN l2_div1 := TRUE;
            ELSE l3_div1 := TRUE; END_IF;
            div_act_1 := div_act_1 + 1;
          END_IF;
          IF obelt = 2 THEN
            IF st_lane[j] = 1 THEN l1_div2 := TRUE;
            ELSIF st_lane[j] = 2 THEN l2_div2 := TRUE;
            ELSE l3_div2 := TRUE; END_IF;
            div_act_2 := div_act_2 + 1;
          END_IF;
          IF obelt = 3 THEN
            IF st_lane[j] = 1 THEN l1_div3 := TRUE;
            ELSIF st_lane[j] = 2 THEN l2_div3 := TRUE;
            ELSE l3_div3 := TRUE; END_IF;
            div_act_3 := div_act_3 + 1;
          END_IF;
        END_IF;
        IF plant_event_actual = 0 OR
           (plant_event_actual >= 1 AND plant_event_actual <= 3 AND
            plant_event_actual = obelt AND st_state[j] = 3) THEN
          st_state[j] := 4;
        ELSE
          plant_fault := 3; sorter_run := FALSE;
        END_IF;
      ELSIF plant_event_type = 4 AND st_state[j] = 4 AND
            plant_event_actual >= 1 AND plant_event_actual <= 9 AND
            (NOT chute_mode OR plant_event_actual <> 2 OR
             chute_view_occupied < 3) THEN
        IF plant_mode AND plant_event_actual = 2 THEN
          chute_accepted_token := plant_event_token;
          chute_accepted_serial := plant_event_serial;
          chute_accepted_event_seq := plant_event_seq;
        END_IF;
        st_actual[j] := plant_event_actual;
        IF st_dest[j] = plant_event_actual THEN
          st_state[j] := 5; st_reason[j] := 0;
        ELSE
          st_state[j] := 7; st_reason[j] := 5;
          missort_ct := missort_ct + 1;
        END_IF;
        IF plant_event_actual = 1 THEN tr11_ct := tr11_ct + 1; END_IF;
        IF plant_event_actual = 2 THEN tr12_ct := tr12_ct + 1; END_IF;
        IF plant_event_actual = 3 THEN tr13_ct := tr13_ct + 1; END_IF;
        IF plant_event_actual = 4 THEN tr21_ct := tr21_ct + 1; END_IF;
        IF plant_event_actual = 5 THEN tr22_ct := tr22_ct + 1; END_IF;
        IF plant_event_actual = 6 THEN tr23_ct := tr23_ct + 1; END_IF;
        IF plant_event_actual = 7 THEN tr31_ct := tr31_ct + 1; END_IF;
        IF plant_event_actual = 8 THEN tr32_ct := tr32_ct + 1; END_IF;
        IF plant_event_actual = 9 THEN tr33_ct := tr33_ct + 1; END_IF;
        IF st_reason[j] = 5 THEN
          IF plant_event_actual = 1 THEN tr11_bad := tr11_bad + 1; END_IF;
          IF plant_event_actual = 2 THEN tr12_bad := tr12_bad + 1; END_IF;
          IF plant_event_actual = 3 THEN tr13_bad := tr13_bad + 1; END_IF;
          IF plant_event_actual = 4 THEN tr21_bad := tr21_bad + 1; END_IF;
          IF plant_event_actual = 5 THEN tr22_bad := tr22_bad + 1; END_IF;
          IF plant_event_actual = 6 THEN tr23_bad := tr23_bad + 1; END_IF;
          IF plant_event_actual = 7 THEN tr31_bad := tr31_bad + 1; END_IF;
          IF plant_event_actual = 8 THEN tr32_bad := tr32_bad + 1; END_IF;
          IF plant_event_actual = 9 THEN tr33_bad := tr33_bad + 1; END_IF;
        END_IF;
      ELSIF plant_event_type = 5 AND st_state[j] >= 1 AND st_state[j] <= 4 THEN
        st_state[j] := 6; st_reason[j] := 1;
        recirc_ct := recirc_ct + 1;
      ELSIF plant_event_type = 6 AND st_state[j] >= 1 AND st_state[j] <= 4 THEN
        st_state[j] := 7; st_reason[j] := 4;
        nohome_ct := nohome_ct + 1; nohome_alarm := TRUE;
        plant_failed_count := plant_failed_count + 1;
        plant_failed_lane := st_lane[j];
      ELSE
        plant_fault := 3; sorter_run := FALSE;
      END_IF;
    ELSE
      plant_fault := 3; sorter_run := FALSE;
    END_IF;
  END_IF;
END_IF;
plant_heartbeat_age := plant_hb_age;
IF NOT plant_mode THEN
  p0_view_status := 0; p1_view_status := 0; p2_view_status := 0;
  p0_view_token := 0; p1_view_token := 0; p2_view_token := 0;
  p0_view_belt := 0; p1_view_belt := 0; p2_view_belt := 0;
END_IF;
slot0_lane := st_lane[0]; slot1_lane := st_lane[1]; slot2_lane := st_lane[2];

(* Accept one command for the current scanned package before cell 14.
   A package without a valid command retains route zero and recirculates. *)
IF xle_mode AND NOT xle_multi AND xle_cmd_id <> 0 AND xle_cmd_id <> xle_cmd_seen THEN
  xle_cmd_seen := xle_cmd_id;
  xle_ack_id := xle_cmd_id;
  xle_state := 4; xle_reason := 2; xle_actual := 0;
  IF xle_cmd_nonce = reset_nonce AND xle_cmd_bc = xle_package AND
     xle_package <> 0 AND xle_cmd_dest >= 1 AND xle_cmd_dest <= 9 THEN
    FOR i := 10 TO 13 DO
      IF ib1[i] = xle_package THEN
        xle_route_dest := xle_cmd_dest;
        obelt := ((xle_route_dest - 1) / 3) + 1;
        IF obelt = 1 THEN rt1[i] := 14;
        ELSIF obelt = 2 THEN rt1[i] := 16;
        ELSE rt1[i] := 18;
        END_IF;
        xle_state := 1; xle_reason := 0;
        xle_accept_tick := scan_ct;
      END_IF;
    END_FOR;
  END_IF;
END_IF;

(* A changed ID commits the complete multi command. All identity fields must
   match one occupied slot; a route is accepted once and only before cell 14.
   Release is separate and valid only after a terminal physical outcome. *)
IF xle_mode AND xle_multi AND multi_cmd_id <> 0 AND multi_cmd_id <> multi_seen THEN
  multi_seen := multi_cmd_id;
  multi_ack := 2;
  multi_ack_id := multi_cmd_id;
  j := multi_slot;
  IF j >= 0 AND j <= 2 THEN
    IF epoch_fault = 0 AND cmd_epoch_lo = epoch_active_lo AND
       cmd_epoch_hi = epoch_active_hi AND multi_nonce = reset_nonce AND st_state[j] <> 0 AND
       multi_token = st_token[j] AND multi_serial = st_serial[j] AND
       multi_seq = st_seq[j] AND multi_bc = st_bc[j] THEN
      IF multi_op = 1 AND xle_liveness = 0 AND hb_ready AND
         hb_age <= 50 AND st_state[j] = 2 AND st_bc[j] <> 0 AND
         multi_dest >= 1 AND multi_dest <= 9 THEN
        FOR i := 10 TO 13 DO
          IF tok1[i] = st_token[j] OR (plant_mode AND i = 10) THEN
            st_dest[j] := multi_dest;
            obelt := ((multi_dest - 1) / 3) + 1;
            IF NOT plant_mode THEN
              IF obelt = 1 THEN rt1[i] := 14;
              ELSIF obelt = 2 THEN rt1[i] := 16;
              ELSE rt1[i] := 18;
              END_IF;
            END_IF;
            st_state[j] := 3; st_accept[j] := scan_ct;
            st_command[j] := multi_cmd_id;
            multi_ack := 1;
          END_IF;
        END_FOR;
      ELSIF multi_op = 2 AND st_state[j] >= 5 THEN
        st_state[j] := 0; st_token[j] := 0; st_lane[j] := 0;
        multi_ack := 3;
      END_IF;
    END_IF;
  END_IF;
END_IF;

(* Three global slots are shared by the three inducts. At each free slot, scan
   ready lanes starting at plant_next_lane and wrap 3 -> 1. A successful
   request advances the pointer. The INDUCT event completes the request
   before another slot may be assigned. *)
IF plant_mode THEN
  IF tmr1 < rate_sp_1 THEN tmr1 := tmr1 + 1; END_IF;
  IF tmr2 < rate_sp_2 THEN tmr2 := tmr2 + 1; END_IF;
  IF tmr3 < rate_sp_3 THEN tmr3 := tmr3 + 1; END_IF;
  IF NOT plant_request_pending AND sorter_run AND plant_fault = 0 AND
     (NOT chute_mode OR chute_quality = 1) AND
     epoch_fault = 0 AND xle_liveness = 0 AND hb_ready AND hb_age <= 50 AND
     (NOT accumulation_mode OR (z_fault = 0 AND z_view_age <= 15)) THEN
    slot_index := -1;
    FOR j := 0 TO 2 DO
      IF st_state[j] = 0 AND slot_index = -1 THEN slot_index := j; END_IF;
    END_FOR;
    IF slot_index >= 0 THEN
      plant_pick_lane := 0;
      FOR i := 0 TO 2 DO
        plant_candidate := ((plant_next_lane - 1 + i) MOD 3) + 1;
        IF plant_pick_lane = 0 AND
           (NOT accumulation_mode OR
            (plant_candidate = 1 AND (z_view_ready MOD 2) = 1) OR
            (plant_candidate = 2 AND ((z_view_ready / 2) MOD 2) = 1) OR
            (plant_candidate = 3 AND ((z_view_ready / 4) MOD 2) = 1)) AND
           ((plant_candidate = 1 AND lane1_run AND tmr1 >= rate_sp_1) OR
            (plant_candidate = 2 AND lane2_run AND tmr2 >= rate_sp_2) OR
            (plant_candidate = 3 AND lane3_run AND tmr3 >= rate_sp_3)) THEN
          plant_pick_lane := plant_candidate;
        END_IF;
      END_FOR;
      IF plant_pick_lane <> 0 THEN
        token_next := token_next + 1;
        IF token_next > 30000 THEN token_next := 1; END_IF;
        st_token[slot_index] := token_next;
        st_lane[slot_index] := plant_pick_lane;
        st_serial[slot_index] := serial_next;
        st_seq[slot_index] := 0; st_bc[slot_index] := 0;
        st_state[slot_index] := 1; st_dest[slot_index] := 0;
        st_actual[slot_index] := 0; st_reason[slot_index] := 0;
        st_scan[slot_index] := 0; st_accept[slot_index] := 0;
        st_divert[slot_index] := 0; st_command[slot_index] := 0;
        plant_request_token := token_next;
        plant_request_serial := serial_next;
        plant_request_lane := plant_pick_lane;
        plant_request := token_next;
        plant_request_pending := TRUE;
        IF plant_pick_lane = 1 THEN tmr1 := 0; END_IF;
        IF plant_pick_lane = 2 THEN tmr2 := 0; END_IF;
        IF plant_pick_lane = 3 THEN tmr3 := 0; END_IF;
        plant_next_lane := (plant_pick_lane MOD 3) + 1;
        serial_next := serial_next + 1;
        IF serial_next > 999 THEN serial_next := 1; END_IF;
      END_IF;
    END_IF;
  END_IF;
END_IF;
